      "I661.6" { ExternalVisible := 'False'} : Bool := FALSE;   // I661.6
      "I661.7" { ExternalVisible := 'False'} : Bool := FALSE;   // I661.7
      "I662.0" { ExternalVisible := 'False'} : Bool := FALSE;   // I662.0
      "I662.1" { ExternalVisible := 'False'} : Bool := FALSE;   // I662.1
      "I662.2" { ExternalVisible := 'False'} : Bool := FALSE;   // I662.2
      "I662.3" { ExternalVisible := 'False'} : Bool := FALSE;   // I662.3
      "I662.4" { ExternalVisible := 'False'} : Bool := FALSE;   // I662.4
      "I662.5" { ExternalVisible := 'False'} : Bool := FALSE;   // I662.5
      "I662.6" { ExternalVisible := 'False'} : Bool := FALSE;   // I662.6
      "I662.7" { ExternalVisible := 'False'} : Bool := FALSE;   // I662.7
      "I663.0" { ExternalVisible := 'False'} : Bool := FALSE;   // I663.0
      "I663.1" { ExternalVisible := 'False'} : Bool := FALSE;   // I663.1
      "I663.2" { ExternalVisible := 'False'} : Bool := FALSE;   // I663.2
      "I663.3" { ExternalVisible := 'False'} : Bool := FALSE;   // I663.3
      "I663.4" { ExternalVisible := 'False'} : Bool := FALSE;   // I663.4
      "I663.5" { ExternalVisible := 'False'} : Bool := FALSE;   // I663.5
      "I663.6" { ExternalVisible := 'False'} : Bool := FALSE;   // I663.6
      "I663.7" { ExternalVisible := 'False'} : Bool := FALSE;   // I663.7
      "I664.0" { ExternalVisible := 'False'} : Bool := FALSE;   // I664.0
      "I664.1" { ExternalVisible := 'False'} : Bool := FALSE;   // I664.1
      "I664.2" { ExternalVisible := 'False'} : Bool := FALSE;   // I664.2
      "I664.3" { ExternalVisible := 'False'} : Bool := FALSE;   // I664.3
      "I664.4" { ExternalVisible := 'False'} : Bool := FALSE;   // I664.4
      "I664.5" { ExternalVisible := 'False'} : Bool := FALSE;   // I664.5
      "I664.6" { ExternalVisible := 'False'} : Bool := FALSE;   // I664.6
      "I664.7" { ExternalVisible := 'False'} : Bool := FALSE;   // I664.7
      "I665.0" { ExternalVisible := 'False'} : Bool := FALSE;   // I665.0
      "I665.1" { ExternalVisible := 'False'} : Bool := FALSE;   // I665.1
      "I665.2" { ExternalVisible := 'False'} : Bool := FALSE;   // I665.2
      "I665.3" { ExternalVisible := 'False'} : Bool := FALSE;   // I665.3
      "I665.4" { ExternalVisible := 'False'} : Bool := FALSE;   // I665.4
      "I665.5" { ExternalVisible := 'False'} : Bool := FALSE;   // I665.5
      "I665.6" { ExternalVisible := 'False'} : Bool := FALSE;   // I665.6
      "I665.7" { ExternalVisible := 'False'} : Bool := FALSE;   // I665.7
      "I666.0" { ExternalVisible := 'False'} : Bool := FALSE;   // I666.0
      "I666.1" { ExternalVisible := 'False'} : Bool := FALSE;   // I666.1
      "I666.2" { ExternalVisible := 'False'} : Bool := FALSE;   // I666.2
      "I666.3" { ExternalVisible := 'False'} : Bool := FALSE;   // I666.3
      "I666.4" { ExternalVisible := 'False'} : Bool := FALSE;   // I666.4
      "I666.5" { ExternalVisible := 'False'} : Bool := FALSE;   // I666.5
      "I666.6" { ExternalVisible := 'False'} : Bool := FALSE;   // I666.6
      "I666.7" { ExternalVisible := 'False'} : Bool := FALSE;   // I666.7
      "I667.0" { ExternalVisible := 'False'} : Bool := FALSE;   // I667.0
      "I667.1" { ExternalVisible := 'False'} : Bool := FALSE;   // I667.1
      "I667.2" { ExternalVisible := 'False'} : Bool := FALSE;   // I667.2
      "I667.3" { ExternalVisible := 'False'} : Bool := FALSE;   // I667.3
      "I667.4" { ExternalVisible := 'False'} : Bool := FALSE;   // I667.4
      "I667.5" { ExternalVisible := 'False'} : Bool := FALSE;   // I667.5
      "I667.6" { ExternalVisible := 'False'} : Bool := FALSE;   // I667.6
      "I667.7" { ExternalVisible := 'False'} : Bool := FALSE;   // I667.7
      "I668.0" { ExternalVisible := 'False'} : Bool := FALSE;   // I668.0
      "I668.1" { ExternalVisible := 'False'} : Bool := FALSE;   // I668.1
      "I668.2" { ExternalVisible := 'False'} : Bool := FALSE;   // I668.2
      "I668.3" { ExternalVisible := 'False'} : Bool := FALSE;   // I668.3
      "I668.4" { ExternalVisible := 'False'} : Bool := FALSE;   // I668.4
      "I668.5" { ExternalVisible := 'False'} : Bool := FALSE;   // I668.5
      "I668.6" { ExternalVisible := 'False'} : Bool := FALSE;   // I668.6
      "I668.7" { ExternalVisible := 'False'} : Bool := FALSE;   // I668.7
      "I669.0" { ExternalVisible := 'False'} : Bool := FALSE;   // I669.0
      "I669.1" { ExternalVisible := 'False'} : Bool := FALSE;   // I669.1
      "I669.2" { ExternalVisible := 'False'} : Bool := FALSE;   // I669.2
      "I669.3" { ExternalVisible := 'False'} : Bool := FALSE;   // I669.3
      "I669.4" { ExternalVisible := 'False'} : Bool := FALSE;   // I669.4
      "I669.5" { ExternalVisible := 'False'} : Bool := FALSE;   // I669.5
      "I669.6" { ExternalVisible := 'False'} : Bool := FALSE;   // I669.6
      "I669.7" { ExternalVisible := 'False'} : Bool := FALSE;   // I669.7
      "I670.0" { ExternalVisible := 'False'} : Bool := FALSE;   // I670.0
      "I670.1" { ExternalVisible := 'False'} : Bool := FALSE;   // I670.1
      "I670.2" { ExternalVisible := 'False'} : Bool := FALSE;   // I670.2
      "I670.3" { ExternalVisible := 'False'} : Bool := FALSE;   // I670.3
      "I670.4" { ExternalVisible := 'False'} : Bool := FALSE;   // I670.4
      "I670.5" { ExternalVisible := 'False'} : Bool := FALSE;   // I670.5
      "I670.6" { ExternalVisible := 'False'} : Bool := FALSE;   // I670.6
      "I670.7" { ExternalVisible := 'False'} : Bool := FALSE;   // I670.7
      "I671.0" { ExternalVisible := 'False'} : Bool := FALSE;   // I671.0
      "I671.1" { ExternalVisible := 'False'} : Bool := FALSE;   // I671.1
      "I671.2" { ExternalVisible := 'False'} : Bool := FALSE;   // I671.2
      "I671.3" { ExternalVisible := 'False'} : Bool := FALSE;   // I671.3
      "I671.4" { ExternalVisible := 'False'} : Bool := FALSE;   // I671.4
      "I671.5" { ExternalVisible := 'False'} : Bool := FALSE;   // I671.5
      "I671.6" { ExternalVisible := 'False'} : Bool := FALSE;   // I671.6
      "I671.7" { ExternalVisible := 'False'} : Bool := FALSE;   // I671.7
      "I672.0" { ExternalVisible := 'False'} : Bool := FALSE;   // I672.0
      "I672.1" { ExternalVisible := 'False'} : Bool := FALSE;   // I672.1
      "I672.2" { ExternalVisible := 'False'} : Bool := FALSE;   // I672.2
      "I672.3" { ExternalVisible := 'False'} : Bool := FALSE;   // I672.3
      "I672.4" { ExternalVisible := 'False'} : Bool := FALSE;   // I672.4
      "I672.5" { ExternalVisible := 'False'} : Bool := FALSE;   // I672.5
      "I672.6" { ExternalVisible := 'False'} : Bool := FALSE;   // I672.6
      "I672.7" { ExternalVisible := 'False'} : Bool := FALSE;   // I672.7
      "I673.0" { ExternalVisible := 'False'} : Bool := FALSE;   // I673.0
      "I673.1" { ExternalVisible := 'False'} : Bool := FALSE;   // I673.1
      "I673.2" { ExternalVisible := 'False'} : Bool := FALSE;   // I673.2
      "I673.3" { ExternalVisible := 'False'} : Bool := FALSE;   // I673.3
      "I673.4" { ExternalVisible := 'False'} : Bool := FALSE;   // I673.4
      "I673.5" { ExternalVisible := 'False'} : Bool := FALSE;   // I673.5
      "I673.6" { ExternalVisible := 'False'} : Bool := FALSE;   // I673.6
      "I673.7" { ExternalVisible := 'False'} : Bool := FALSE;   // I673.7
      "I674.0" { ExternalVisible := 'False'} : Bool := FALSE;   // I674.0
      "I674.1" { ExternalVisible := 'False'} : Bool := FALSE;   // I674.1
      "I674.2" { ExternalVisible := 'False'} : Bool := FALSE;   // I674.2
      "I674.3" { ExternalVisible := 'False'} : Bool := FALSE;   // I674.3
      "I674.4" { ExternalVisible := 'False'} : Bool := FALSE;   // I674.4
      "I674.5" { ExternalVisible := 'False'} : Bool := FALSE;   // I674.5
      "I674.6" { ExternalVisible := 'False'} : Bool := FALSE;   // I674.6
      "I674.7" { ExternalVisible := 'False'} : Bool := FALSE;   // I674.7
      "I675.0" { ExternalVisible := 'False'} : Bool := FALSE;   // I675.0
      "I675.1" { ExternalVisible := 'False'} : Bool := FALSE;   // I675.1
      "I675.2" { ExternalVisible := 'False'} : Bool := FALSE;   // I675.2
      "I675.3" { ExternalVisible := 'False'} : Bool := FALSE;   // I675.3
      "I675.4" { ExternalVisible := 'False'} : Bool := FALSE;   // I675.4
      "I675.5" { ExternalVisible := 'False'} : Bool := FALSE;   // I675.5
      "I675.6" { ExternalVisible := 'False'} : Bool := FALSE;   // I675.6
      "I675.7" { ExternalVisible := 'False'} : Bool := FALSE;   // I675.7
      "I676.0" { ExternalVisible := 'False'} : Bool := FALSE;   // I676.0
      "I676.1" { ExternalVisible := 'False'} : Bool := FALSE;   // I676.1
      "I676.2" { ExternalVisible := 'False'} : Bool := FALSE;   // I676.2
      "I676.3" { ExternalVisible := 'False'} : Bool := FALSE;   // I676.3
      "I676.4" { ExternalVisible := 'False'} : Bool := FALSE;   // I676.4
      "I676.5" { ExternalVisible := 'False'} : Bool := FALSE;   // I676.5
      "I676.6" { ExternalVisible := 'False'} : Bool := FALSE;   // I676.6
      "I676.7" { ExternalVisible := 'False'} : Bool := FALSE;   // I676.7
      "I677.0" { ExternalVisible := 'False'} : Bool := FALSE;   // I677.0
      "I677.1" { ExternalVisible := 'False'} : Bool := FALSE;   // I677.1
      "I677.2" { ExternalVisible := 'False'} : Bool := FALSE;   // I677.2
      "I677.3" { ExternalVisible := 'False'} : Bool := FALSE;   // I677.3
      "I677.4" { ExternalVisible := 'False'} : Bool := FALSE;   // I677.4
      "I677.5" { ExternalVisible := 'False'} : Bool := FALSE;   // I677.5
      "I677.6" { ExternalVisible := 'False'} : Bool := FALSE;   // I677.6
      "I677.7" { ExternalVisible := 'False'} : Bool := FALSE;   // I677.7
      "I678.0" { ExternalVisible := 'False'} : Bool := FALSE;   // I678.0
      "I678.1" { ExternalVisible := 'False'} : Bool := FALSE;   // I678.1
      "I678.2" { ExternalVisible := 'False'} : Bool := FALSE;   // I678.2
      "I678.3" { ExternalVisible := 'False'} : Bool := FALSE;   // I678.3
      "I678.4" { ExternalVisible := 'False'} : Bool := FALSE;   // I678.4
      "I678.5" { ExternalVisible := 'False'} : Bool := FALSE;   // I678.5
      "I678.6" { ExternalVisible := 'False'} : Bool := FALSE;   // I678.6
      "I678.7" { ExternalVisible := 'False'} : Bool := FALSE;   // I678.7
      "I679.0" { ExternalVisible := 'False'} : Bool := FALSE;   // I679.0
      "I679.1" { ExternalVisible := 'False'} : Bool := FALSE;   // I679.1
      "I679.2" { ExternalVisible := 'False'} : Bool := FALSE;   // I679.2
      "I679.3" { ExternalVisible := 'False'} : Bool := FALSE;   // I679.3
      "I679.4" { ExternalVisible := 'False'} : Bool := FALSE;   // I679.4
      "I679.5" { ExternalVisible := 'False'} : Bool := FALSE;   // I679.5
      "I679.6" { ExternalVisible := 'False'} : Bool := FALSE;   // I679.6
      "I679.7" { ExternalVisible := 'False'} : Bool := FALSE;   // I679.7
      "I680.0" { ExternalVisible := 'False'} : Bool := FALSE;   // I680.0
      "I680.1" { ExternalVisible := 'False'} : Bool := FALSE;   // I680.1
      "I680.2" { ExternalVisible := 'False'} : Bool := FALSE;   // I680.2
      "I680.3" { ExternalVisible := 'False'} : Bool := FALSE;   // I680.3
      "I680.4" { ExternalVisible := 'False'} : Bool := FALSE;   // I680.4
      "I680.5" { ExternalVisible := 'False'} : Bool := FALSE;   // I680.5
      "I680.6" { ExternalVisible := 'False'} : Bool := FALSE;   // I680.6
      "I680.7" { ExternalVisible := 'False'} : Bool := FALSE;   // I680.7
      "I681.0" { ExternalVisible := 'False'} : Bool := FALSE;   // I681.0
      "I681.1" { ExternalVisible := 'False'} : Bool := FALSE;   // I681.1
      "I681.2" { ExternalVisible := 'False'} : Bool := FALSE;   // I681.2
      "I681.3" { ExternalVisible := 'False'} : Bool := FALSE;   // I681.3
      "I681.4" { ExternalVisible := 'False'} : Bool := FALSE;   // I681.4
      "I681.5" { ExternalVisible := 'False'} : Bool := FALSE;   // I681.5
      "I681.6" { ExternalVisible := 'False'} : Bool := FALSE;   // I681.6
      "I681.7" { ExternalVisible := 'False'} : Bool := FALSE;   // I681.7
      "I682.0" { ExternalVisible := 'False'} : Bool := FALSE;   // I682.0
      "I682.1" { ExternalVisible := 'False'} : Bool := FALSE;   // I682.1
      "I682.2" { ExternalVisible := 'False'} : Bool := FALSE;   // I682.2
      "I682.3" { ExternalVisible := 'False'} : Bool := FALSE;   // I682.3
      "I682.4" { ExternalVisible := 'False'} : Bool := FALSE;   // I682.4
      "I682.5" { ExternalVisible := 'False'} : Bool := FALSE;   // I682.5
      "I682.6" { ExternalVisible := 'False'} : Bool := FALSE;   // I682.6
      "I682.7" { ExternalVisible := 'False'} : Bool := FALSE;   // I682.7
      "I683.0" { ExternalVisible := 'False'} : Bool := FALSE;   // I683.0
      "I683.1" { ExternalVisible := 'False'} : Bool := FALSE;   // I683.1
      "I683.2" { ExternalVisible := 'False'} : Bool := FALSE;   // I683.2
      "I683.3" { ExternalVisible := 'False'} : Bool := FALSE;   // I683.3
      "I683.4" { ExternalVisible := 'False'} : Bool := FALSE;   // I683.4
      "I683.5" { ExternalVisible := 'False'} : Bool := FALSE;   // I683.5
      "I683.6" { ExternalVisible := 'False'} : Bool := FALSE;   // I683.6
      "I683.7" { ExternalVisible := 'False'} : Bool := FALSE;   // I683.7
      "I684.0" { ExternalVisible := 'False'} : Bool := FALSE;   // I684.0
      "I684.1" { ExternalVisible := 'False'} : Bool := FALSE;   // I684.1
      "I684.2" { ExternalVisible := 'False'} : Bool := FALSE;   // I684.2
      "I684.3" { ExternalVisible := 'False'} : Bool := FALSE;   // I684.3
      "I684.4" { ExternalVisible := 'False'} : Bool := FALSE;   // I684.4
      "I684.5" { ExternalVisible := 'False'} : Bool := FALSE;   // I684.5
      "I684.6" { ExternalVisible := 'False'} : Bool := FALSE;   // I684.6
      "I684.7" { ExternalVisible := 'False'} : Bool := FALSE;   // I684.7
      "I685.0" { ExternalVisible := 'False'} : Bool := FALSE;   // I685.0
      "I685.1" { ExternalVisible := 'False'} : Bool := FALSE;   // I685.1
      "I685.2" { ExternalVisible := 'False'} : Bool := FALSE;   // I685.2
      "I685.3" { ExternalVisible := 'False'} : Bool := FALSE;   // I685.3
      "I685.4" { ExternalVisible := 'False'} : Bool := FALSE;   // I685.4
      "I685.5" { ExternalVisible := 'False'} : Bool := FALSE;   // I685.5
      "I685.6" { ExternalVisible := 'False'} : Bool := FALSE;   // I685.6
      "I685.7" { ExternalVisible := 'False'} : Bool := FALSE;   // I685.7
      "I686.0" { ExternalVisible := 'False'} : Bool := FALSE;   // I686.0
      "I686.1" { ExternalVisible := 'False'} : Bool := FALSE;   // I686.1
      "I686.2" { ExternalVisible := 'False'} : Bool := FALSE;   // I686.2
      "I686.3" { ExternalVisible := 'False'} : Bool := FALSE;   // I686.3
      "I686.4" { ExternalVisible := 'False'} : Bool := FALSE;   // I686.4
      "I686.5" { ExternalVisible := 'False'} : Bool := FALSE;   // I686.5
      "I686.6" { ExternalVisible := 'False'} : Bool := FALSE;   // I686.6
      "I686.7" { ExternalVisible := 'False'} : Bool := FALSE;   // I686.7
      "I687.0" { ExternalVisible := 'False'} : Bool := FALSE;   // I687.0
      "I687.1" { ExternalVisible := 'False'} : Bool := FALSE;   // I687.1
      "I687.2" { ExternalVisible := 'False'} : Bool := FALSE;   // I687.2
      "I687.3" { ExternalVisible := 'False'} : Bool := FALSE;   // I687.3
      "I687.4" { ExternalVisible := 'False'} : Bool := FALSE;   // I687.4
      "I687.5" { ExternalVisible := 'False'} : Bool := FALSE;   // I687.5
      "I687.6" { ExternalVisible := 'False'} : Bool := FALSE;   // I687.6
      "I687.7" { ExternalVisible := 'False'} : Bool := FALSE;   // I687.7
      "I688.0" { ExternalVisible := 'False'} : Bool := FALSE;   // I688.0
      "I688.1" { ExternalVisible := 'False'} : Bool := FALSE;   // I688.1
      "I688.2" { ExternalVisible := 'False'} : Bool := FALSE;   // I688.2
      "I688.3" { ExternalVisible := 'False'} : Bool := FALSE;   // I688.3
      "I688.4" { ExternalVisible := 'False'} : Bool := FALSE;   // I688.4
      "I688.5" { ExternalVisible := 'False'} : Bool := FALSE;   // I688.5
      "I688.6" { ExternalVisible := 'False'} : Bool := FALSE;   // I688.6
      "I688.7" { ExternalVisible := 'False'} : Bool := FALSE;   // I688.7
      "I689.0" { ExternalVisible := 'False'} : Bool := FALSE;   // I689.0
      "I689.1" { ExternalVisible := 'False'} : Bool := FALSE;   // I689.1
      "I689.2" { ExternalVisible := 'False'} : Bool := FALSE;   // I689.2
      "I689.3" { ExternalVisible := 'False'} : Bool := FALSE;   // I689.3
      "I689.4" { ExternalVisible := 'False'} : Bool := FALSE;   // I689.4
      "I689.5" { ExternalVisible := 'False'} : Bool := FALSE;   // I689.5
      "I689.6" { ExternalVisible := 'False'} : Bool := FALSE;   // I689.6
      "I689.7" { ExternalVisible := 'False'} : Bool := FALSE;   // I689.7
      "I690.0" { ExternalVisible := 'False'} : Bool := FALSE;   // I690.0
      "I690.1" { ExternalVisible := 'False'} : Bool := FALSE;   // I690.1
      "I690.2" { ExternalVisible := 'False'} : Bool := FALSE;   // I690.2
      "I690.3" { ExternalVisible := 'False'} : Bool := FALSE;   // I690.3
      "I690.4" { ExternalVisible := 'False'} : Bool := FALSE;   // I690.4
      "I690.5" { ExternalVisible := 'False'} : Bool := FALSE;   // I690.5
      "I690.6" { ExternalVisible := 'False'} : Bool := FALSE;   // I690.6
      "I690.7" { ExternalVisible := 'False'} : Bool := FALSE;   // I690.7
      "I691.0" { ExternalVisible := 'False'} : Bool := FALSE;   // I691.0
      "I691.1" { ExternalVisible := 'False'} : Bool := FALSE;   // I691.1
      "I691.2" { ExternalVisible := 'False'} : Bool := FALSE;   // I691.2
      "I691.3" { ExternalVisible := 'False'} : Bool := FALSE;   // I691.3
      "I691.4" { ExternalVisible := 'False'} : Bool := FALSE;   // I691.4
      "I691.5" { ExternalVisible := 'False'} : Bool := FALSE;   // I691.5
      "I691.6" { ExternalVisible := 'False'} : Bool := FALSE;   // I691.6
      "I691.7" { ExternalVisible := 'False'} : Bool := FALSE;   // I691.7
      "I692.0" { ExternalVisible := 'False'} : Bool := FALSE;   // I692.0
      "I692.1" { ExternalVisible := 'False'} : Bool := FALSE;   // I692.1
      "I692.2" { ExternalVisible := 'False'} : Bool := FALSE;   // I692.2
      "I692.3" { ExternalVisible := 'False'} : Bool := FALSE;   // I692.3
      "I692.4" { ExternalVisible := 'False'} : Bool := FALSE;   // I692.4
      "I692.5" { ExternalVisible := 'False'} : Bool := FALSE;   // I692.5
      "I692.6" { ExternalVisible := 'False'} : Bool := FALSE;   // I692.6
      "I692.7" { ExternalVisible := 'False'} : Bool := FALSE;   // I692.7
      "I693.0" { ExternalVisible := 'False'} : Bool := FALSE;   // I693.0
      "I693.1" { ExternalVisible := 'False'} : Bool := FALSE;   // I693.1
      "I693.2" { ExternalVisible := 'False'} : Bool := FALSE;   // I693.2
      "I693.3" { ExternalVisible := 'False'} : Bool := FALSE;   // I693.3
      "I693.4" { ExternalVisible := 'False'} : Bool := FALSE;   // I693.4
      "I693.5" { ExternalVisible := 'False'} : Bool := FALSE;   // I693.5
      "I693.6" { ExternalVisible := 'False'} : Bool := FALSE;   // I693.6
      "I693.7" { ExternalVisible := 'False'} : Bool := FALSE;   // I693.7
      "I694.0" { ExternalVisible := 'False'} : Bool := FALSE;   // I694.0
      "I694.1" { ExternalVisible := 'False'} : Bool := FALSE;   // I694.1
      "I694.2" { ExternalVisible := 'False'} : Bool := FALSE;   // I694.2
      "I694.3" { ExternalVisible := 'False'} : Bool := FALSE;   // I694.3
      "I694.4" { ExternalVisible := 'False'} : Bool := FALSE;   // I694.4
      "I694.5" { ExternalVisible := 'False'} : Bool := FALSE;   // I694.5
      "I694.6" { ExternalVisible := 'False'} : Bool := FALSE;   // I694.6
      "I694.7" { ExternalVisible := 'False'} : Bool := FALSE;   // I694.7
      "I695.0" { ExternalVisible := 'False'} : Bool := FALSE;   // I695.0
      "I695.1" { ExternalVisible := 'False'} : Bool := FALSE;   // I695.1
      "I695.2" { ExternalVisible := 'False'} : Bool := FALSE;   // I695.2
      "I695.3" { ExternalVisible := 'False'} : Bool := FALSE;   // I695.3
      "I695.4" { ExternalVisible := 'False'} : Bool := FALSE;   // I695.4
      "I695.5" { ExternalVisible := 'False'} : Bool := FALSE;   // I695.5
      "I695.6" { ExternalVisible := 'False'} : Bool := FALSE;   // I695.6
      "I695.7" { ExternalVisible := 'False'} : Bool := FALSE;   // I695.7
      "I696.0" { ExternalVisible := 'False'} : Bool := FALSE;   // I696.0
      "I696.1" { ExternalVisible := 'False'} : Bool := FALSE;   // I696.1
      "I696.2" { ExternalVisible := 'False'} : Bool := FALSE;   // I696.2
      "I696.3" { ExternalVisible := 'False'} : Bool := FALSE;   // I696.3
      "I696.4" { ExternalVisible := 'False'} : Bool := FALSE;   // I696.4
      "I696.5" { ExternalVisible := 'False'} : Bool := FALSE;   // I696.5
      "I696.6" { ExternalVisible := 'False'} : Bool := FALSE;   // I696.6
      "I696.7" { ExternalVisible := 'False'} : Bool := FALSE;   // I696.7
      "I697.0" { ExternalVisible := 'False'} : Bool := FALSE;   // I697.0
      "I697.1" { ExternalVisible := 'False'} : Bool := FALSE;   // I697.1
      "I697.2" { ExternalVisible := 'False'} : Bool := FALSE;   // I697.2
      "I697.3" { ExternalVisible := 'False'} : Bool := FALSE;   // I697.3
      "I697.4" { ExternalVisible := 'False'} : Bool := FALSE;   // I697.4
      "I697.5" { ExternalVisible := 'False'} : Bool := FALSE;   // I697.5
      "I697.6" { ExternalVisible := 'False'} : Bool := FALSE;   // I697.6
      "I697.7" { ExternalVisible := 'False'} : Bool := FALSE;   // I697.7
      "I698.0" { ExternalVisible := 'False'} : Bool := FALSE;   // I698.0
      "I698.1" { ExternalVisible := 'False'} : Bool := FALSE;   // I698.1
      "I698.2" { ExternalVisible := 'False'} : Bool := FALSE;   // I698.2
      "I698.3" { ExternalVisible := 'False'} : Bool := FALSE;   // I698.3
      "I698.4" { ExternalVisible := 'False'} : Bool := FALSE;   // I698.4
      "I698.5" { ExternalVisible := 'False'} : Bool := FALSE;   // I698.5
      "I698.6" { ExternalVisible := 'False'} : Bool := FALSE;   // I698.6
      "I698.7" { ExternalVisible := 'False'} : Bool := FALSE;   // I698.7
      "I699.0" { ExternalVisible := 'False'} : Bool := FALSE;   // I699.0
      "I699.1" { ExternalVisible := 'False'} : Bool := FALSE;   // I699.1
      "I699.2" { ExternalVisible := 'False'} : Bool := FALSE;   // I699.2
      "I699.3" { ExternalVisible := 'False'} : Bool := FALSE;   // I699.3
      "I699.4" { ExternalVisible := 'False'} : Bool := FALSE;   // I699.4
      "I699.5" { ExternalVisible := 'False'} : Bool := FALSE;   // I699.5
      "I699.6" { ExternalVisible := 'False'} : Bool := FALSE;   // I699.6
      "I699.7" { ExternalVisible := 'False'} : Bool := FALSE;   // I699.7
      "I700.0" { ExternalVisible := 'False'} : Bool := FALSE;   // I700.0
      "I700.1" { ExternalVisible := 'False'} : Bool := FALSE;   // I700.1
      "I700.2" { ExternalVisible := 'False'} : Bool := FALSE;   // I700.2
      "I700.3" { ExternalVisible := 'False'} : Bool := FALSE;   // I700.3
      "I700.4" { ExternalVisible := 'False'} : Bool := FALSE;   // I700.4
      "I700.5" { ExternalVisible := 'False'} : Bool := FALSE;   // I700.5
      "I700.6" { ExternalVisible := 'False'} : Bool := FALSE;   // I700.6
      "I700.7" { ExternalVisible := 'False'} : Bool := FALSE;   // I700.7
      "I701.0" { ExternalVisible := 'False'} : Bool := FALSE;   // I701.0
      "I701.1" { ExternalVisible := 'False'} : Bool := FALSE;   // I701.1
      "I701.2" { ExternalVisible := 'False'} : Bool := FALSE;   // I701.2
      "I701.3" { ExternalVisible := 'False'} : Bool := FALSE;   // I701.3
      "I701.4" { ExternalVisible := 'False'} : Bool := FALSE;   // I701.4
      "I701.5" { ExternalVisible := 'False'} : Bool := FALSE;   // I701.5
      "I701.6" { ExternalVisible := 'False'} : Bool := FALSE;   // I701.6
      "I701.7" { ExternalVisible := 'False'} : Bool := FALSE;   // I701.7
      "I702.0" { ExternalVisible := 'False'} : Bool := FALSE;   // I702.0
      "I702.1" { ExternalVisible := 'False'} : Bool := FALSE;   // I702.1
      "I702.2" { ExternalVisible := 'False'} : Bool := FALSE;   // I702.2
      "I702.3" { ExternalVisible := 'False'} : Bool := FALSE;   // I702.3
      "I702.4" { ExternalVisible := 'False'} : Bool := FALSE;   // I702.4
      "I702.5" { ExternalVisible := 'False'} : Bool := FALSE;   // I702.5
      "I702.6" { ExternalVisible := 'False'} : Bool := FALSE;   // I702.6
      "I702.7" { ExternalVisible := 'False'} : Bool := FALSE;   // I702.7
      "I703.0" { ExternalVisible := 'False'} : Bool := FALSE;   // I703.0
      "I703.1" { ExternalVisible := 'False'} : Bool := FALSE;   // I703.1
      "I703.2" { ExternalVisible := 'False'} : Bool := FALSE;   // I703.2
      "I703.3" { ExternalVisible := 'False'} : Bool := FALSE;   // I703.3
      "I703.4" { ExternalVisible := 'False'} : Bool := FALSE;   // I703.4
      "I703.5" { ExternalVisible := 'False'} : Bool := FALSE;   // I703.5
      "I703.6" { ExternalVisible := 'False'} : Bool := FALSE;   // I703.6
      "I703.7" { ExternalVisible := 'False'} : Bool := FALSE;   // I703.7
      "I704.0" { ExternalVisible := 'False'} : Bool := FALSE;   // I704.0
      "I704.1" { ExternalVisible := 'False'} : Bool := FALSE;   // I704.1
      "I704.2" { ExternalVisible := 'False'} : Bool := FALSE;   // I704.2
      "I704.3" { ExternalVisible := 'False'} : Bool := FALSE;   // I704.3
      "I704.4" { ExternalVisible := 'False'} : Bool := FALSE;   // I704.4
      "I704.5" { ExternalVisible := 'False'} : Bool := FALSE;   // I704.5
      "I704.6" { ExternalVisible := 'False'} : Bool := FALSE;   // I704.6
      "I704.7" { ExternalVisible := 'False'} : Bool := FALSE;   // I704.7
      "I705.0" { ExternalVisible := 'False'} : Bool := FALSE;   // I705.0
      "I705.1" { ExternalVisible := 'False'} : Bool := FALSE;   // I705.1
      "I705.2" { ExternalVisible := 'False'} : Bool := FALSE;   // I705.2
      "I705.3" { ExternalVisible := 'False'} : Bool := FALSE;   // I705.3
      "I705.4" { ExternalVisible := 'False'} : Bool := FALSE;   // I705.4
      "I705.5" { ExternalVisible := 'False'} : Bool := FALSE;   // I705.5
      "I705.6" { ExternalVisible := 'False'} : Bool := FALSE;   // I705.6
      "I705.7" { ExternalVisible := 'False'} : Bool := FALSE;   // I705.7
      "I706.0" { ExternalVisible := 'False'} : Bool := FALSE;   // I706.0
      "I706.1" { ExternalVisible := 'False'} : Bool := FALSE;   // I706.1
      "I706.2" { ExternalVisible := 'False'} : Bool := FALSE;   // I706.2
      "I706.3" { ExternalVisible := 'False'} : Bool := FALSE;   // I706.3
      "I706.4" { ExternalVisible := 'False'} : Bool := FALSE;   // I706.4
      "I706.5" { ExternalVisible := 'False'} : Bool := FALSE;   // I706.5
      "I706.6" { ExternalVisible := 'False'} : Bool := FALSE;   // I706.6
      "I706.7" { ExternalVisible := 'False'} : Bool := FALSE;   // I706.7
      "I707.0" { ExternalVisible := 'False'} : Bool := FALSE;   // I707.0
      "I707.1" { ExternalVisible := 'False'} : Bool := FALSE;   // I707.1
      "I707.2" { ExternalVisible := 'False'} : Bool := FALSE;   // I707.2
      "I707.3" { ExternalVisible := 'False'} : Bool := FALSE;   // I707.3
      "I707.4" { ExternalVisible := 'False'} : Bool := FALSE;   // I707.4
      "I707.5" { ExternalVisible := 'False'} : Bool := FALSE;   // I707.5
      "I707.6" { ExternalVisible := 'False'} : Bool := FALSE;   // I707.6
      "I707.7" { ExternalVisible := 'False'} : Bool := FALSE;   // I707.7
      "I708.0" { ExternalVisible := 'False'} : Bool := FALSE;   // I708.0
      "I708.1" { ExternalVisible := 'False'} : Bool := FALSE;   // I708.1
      "I708.2" { ExternalVisible := 'False'} : Bool := FALSE;   // I708.2
      "I708.3" { ExternalVisible := 'False'} : Bool := FALSE;   // I708.3
      "I708.4" { ExternalVisible := 'False'} : Bool := FALSE;   // I708.4
      "I708.5" { ExternalVisible := 'False'} : Bool := FALSE;   // I708.5
      "I708.6" { ExternalVisible := 'False'} : Bool := FALSE;   // I708.6
      "I708.7" { ExternalVisible := 'False'} : Bool := FALSE;   // I708.7
      "I709.0" { ExternalVisible := 'False'} : Bool := FALSE;   // I709.0
      "I709.1" { ExternalVisible := 'False'} : Bool := FALSE;   // I709.1
      "I709.2" { ExternalVisible := 'False'} : Bool := FALSE;   // I709.2
      "I709.3" { ExternalVisible := 'False'} : Bool := FALSE;   // I709.3
      "I709.4" { ExternalVisible := 'False'} : Bool := FALSE;   // I709.4
      "I709.5" { ExternalVisible := 'False'} : Bool := FALSE;   // I709.5
      "I709.6" { ExternalVisible := 'False'} : Bool := FALSE;   // I709.6
      "I709.7" { ExternalVisible := 'False'} : Bool := FALSE;   // I709.7
      "I710.0" { ExternalVisible := 'False'} : Bool := FALSE;   // I710.0
      "I710.1" { ExternalVisible := 'False'} : Bool := FALSE;   // I710.1
      "I710.2" { ExternalVisible := 'False'} : Bool := FALSE;   // I710.2
      "I710.3" { ExternalVisible := 'False'} : Bool := FALSE;   // I710.3
      "I710.4" { ExternalVisible := 'False'} : Bool := FALSE;   // I710.4
      "I710.5" { ExternalVisible := 'False'} : Bool := FALSE;   // I710.5
      "I710.6" { ExternalVisible := 'False'} : Bool := FALSE;   // I710.6
      "I710.7" { ExternalVisible := 'False'} : Bool := FALSE;   // I710.7
      "I711.0" { ExternalVisible := 'False'} : Bool := FALSE;   // I711.0
      "I711.1" { ExternalVisible := 'False'} : Bool := FALSE;   // I711.1
      "I711.2" { ExternalVisible := 'False'} : Bool := FALSE;   // I711.2
      "I711.3" { ExternalVisible := 'False'} : Bool := FALSE;   // I711.3
      "I711.4" { ExternalVisible := 'False'} : Bool := FALSE;   // I711.4
      "I711.5" { ExternalVisible := 'False'} : Bool := FALSE;   // I711.5
      "I711.6" { ExternalVisible := 'False'} : Bool := FALSE;   // I711.6
      "I711.7" { ExternalVisible := 'False'} : Bool := FALSE;   // I711.7
      "I712.0" { ExternalVisible := 'False'} : Bool := FALSE;   // I712.0
      "I712.1" { ExternalVisible := 'False'} : Bool := FALSE;   // I712.1
      "I712.2" { ExternalVisible := 'False'} : Bool := FALSE;   // I712.2
      "I712.3" { ExternalVisible := 'False'} : Bool := FALSE;   // I712.3
      "I712.4" { ExternalVisible := 'False'} : Bool := FALSE;   // I712.4
      "I712.5" { ExternalVisible := 'False'} : Bool := FALSE;   // I712.5
      "I712.6" { ExternalVisible := 'False'} : Bool := FALSE;   // I712.6
      "I712.7" { ExternalVisible := 'False'} : Bool := FALSE;   // I712.7
      "I713.0" { ExternalVisible := 'False'} : Bool := FALSE;   // I713.0
      "I713.1" { ExternalVisible := 'False'} : Bool := FALSE;   // I713.1
      "I713.2" { ExternalVisible := 'False'} : Bool := FALSE;   // I713.2
      "I713.3" { ExternalVisible := 'False'} : Bool := FALSE;   // I713.3
      "I713.4" { ExternalVisible := 'False'} : Bool := FALSE;   // I713.4
      "I713.5" { ExternalVisible := 'False'} : Bool := FALSE;   // I713.5
      "I713.6" { ExternalVisible := 'False'} : Bool := FALSE;   // I713.6
      "I713.7" { ExternalVisible := 'False'} : Bool := FALSE;   // I713.7
      "I714.0" { ExternalVisible := 'False'} : Bool := FALSE;   // I714.0
      "I714.1" { ExternalVisible := 'False'} : Bool := FALSE;   // I714.1
      "I714.2" { ExternalVisible := 'False'} : Bool := FALSE;   // I714.2
      "I714.3" { ExternalVisible := 'False'} : Bool := FALSE;   // I714.3
      "I714.4" { ExternalVisible := 'False'} : Bool := FALSE;   // I714.4
      "I714.5" { ExternalVisible := 'False'} : Bool := FALSE;   // I714.5
      "I714.6" { ExternalVisible := 'False'} : Bool := FALSE;   // I714.6
      "I714.7" { ExternalVisible := 'False'} : Bool := FALSE;   // I714.7
      "I715.0" { ExternalVisible := 'False'} : Bool := FALSE;   // I715.0
      "I715.1" { ExternalVisible := 'False'} : Bool := FALSE;   // I715.1
      "I715.2" { ExternalVisible := 'False'} : Bool := FALSE;   // I715.2
      "I715.3" { ExternalVisible := 'False'} : Bool := FALSE;   // I715.3
      "I715.4" { ExternalVisible := 'False'} : Bool := FALSE;   // I715.4
      "I715.5" { ExternalVisible := 'False'} : Bool := FALSE;   // I715.5
      "I715.6" { ExternalVisible := 'False'} : Bool := FALSE;   // I715.6
      "I715.7" { ExternalVisible := 'False'} : Bool := FALSE;   // I715.7
      "I716.0" { ExternalVisible := 'False'} : Bool := FALSE;   // I716.0
      "I716.1" { ExternalVisible := 'False'} : Bool := FALSE;   // I716.1
      "I716.2" { ExternalVisible := 'False'} : Bool := FALSE;   // I716.2
      "I716.3" { ExternalVisible := 'False'} : Bool := FALSE;   // I716.3
      "I716.4" { ExternalVisible := 'False'} : Bool := FALSE;   // I716.4
      "I716.5" { ExternalVisible := 'False'} : Bool := FALSE;   // I716.5
      "I716.6" { ExternalVisible := 'False'} : Bool := FALSE;   // I716.6
      "I716.7" { ExternalVisible := 'False'} : Bool := FALSE;   // I716.7
      "I717.0" { ExternalVisible := 'False'} : Bool := FALSE;   // I717.0
      "I717.1" { ExternalVisible := 'False'} : Bool := FALSE;   // I717.1
      "I717.2" { ExternalVisible := 'False'} : Bool := FALSE;   // I717.2
      "I717.3" { ExternalVisible := 'False'} : Bool := FALSE;   // I717.3
      "I717.4" { ExternalVisible := 'False'} : Bool := FALSE;   // I717.4
      "I717.5" { ExternalVisible := 'False'} : Bool := FALSE;   // I717.5
      "I717.6" { ExternalVisible := 'False'} : Bool := FALSE;   // I717.6
      "I717.7" { ExternalVisible := 'False'} : Bool := FALSE;   // I717.7
      "I718.0" { ExternalVisible := 'False'} : Bool := FALSE;   // I718.0
      "I718.1" { ExternalVisible := 'False'} : Bool := FALSE;   // I718.1
      "I718.2" { ExternalVisible := 'False'} : Bool := FALSE;   // I718.2
      "I718.3" { ExternalVisible := 'False'} : Bool := FALSE;   // I718.3
      "I718.4" { ExternalVisible := 'False'} : Bool := FALSE;   // I718.4
      "I718.5" { ExternalVisible := 'False'} : Bool := FALSE;   // I718.5
      "I718.6" { ExternalVisible := 'False'} : Bool := FALSE;   // I718.6
      "I718.7" { ExternalVisible := 'False'} : Bool := FALSE;   // I718.7
      "I719.0" { ExternalVisible := 'False'} : Bool := FALSE;   // I719.0
      "I719.1" { ExternalVisible := 'False'} : Bool := FALSE;   // I719.1
      "I719.2" { ExternalVisible := 'False'} : Bool := FALSE;   // I719.2
      "I719.3" { ExternalVisible := 'False'} : Bool := FALSE;   // I719.3
      "I719.4" { ExternalVisible := 'False'} : Bool := FALSE;   // I719.4
      "I719.5" { ExternalVisible := 'False'} : Bool := FALSE;   // I719.5
      "I719.6" { ExternalVisible := 'False'} : Bool := FALSE;   // I719.6
      "I719.7" { ExternalVisible := 'False'} : Bool := FALSE;   // I719.7
      "I720.0" { ExternalVisible := 'False'} : Bool := FALSE;   // I720.0
      "I720.1" { ExternalVisible := 'False'} : Bool := FALSE;   // I720.1
      "I720.2" { ExternalVisible := 'False'} : Bool := FALSE;   // I720.2
      "I720.3" { ExternalVisible := 'False'} : Bool := FALSE;   // I720.3
      "I720.4" { ExternalVisible := 'False'} : Bool := FALSE;   // I720.4
      "I720.5" { ExternalVisible := 'False'} : Bool := FALSE;   // I720.5
      "I720.6" { ExternalVisible := 'False'} : Bool := FALSE;   // I720.6
      "I720.7" { ExternalVisible := 'False'} : Bool := FALSE;   // I720.7
      "I721.0" { ExternalVisible := 'False'} : Bool := FALSE;   // I721.0
      "I721.1" { ExternalVisible := 'False'} : Bool := FALSE;   // I721.1
      "I721.2" { ExternalVisible := 'False'} : Bool := FALSE;   // I721.2
      "I721.3" { ExternalVisible := 'False'} : Bool := FALSE;   // I721.3
      "I721.4" { ExternalVisible := 'False'} : Bool := FALSE;   // I721.4
      "I721.5" { ExternalVisible := 'False'} : Bool := FALSE;   // I721.5
      "I721.6" { ExternalVisible := 'False'} : Bool := FALSE;   // I721.6
      "I721.7" { ExternalVisible := 'False'} : Bool := FALSE;   // I721.7
      "I722.0" { ExternalVisible := 'False'} : Bool := FALSE;   // I722.0
      "I722.1" { ExternalVisible := 'False'} : Bool := FALSE;   // I722.1
      "I722.2" { ExternalVisible := 'False'} : Bool := FALSE;   // I722.2
      "I722.3" { ExternalVisible := 'False'} : Bool := FALSE;   // I722.3
      "I722.4" { ExternalVisible := 'False'} : Bool := FALSE;   // I722.4
      "I722.5" { ExternalVisible := 'False'} : Bool := FALSE;   // I722.5
      "I722.6" { ExternalVisible := 'False'} : Bool := FALSE;   // I722.6
      "I722.7" { ExternalVisible := 'False'} : Bool := FALSE;   // I722.7
      "I723.0" { ExternalVisible := 'False'} : Bool := FALSE;   // I723.0
      "I723.1" { ExternalVisible := 'False'} : Bool := FALSE;   // I723.1
      "I723.2" { ExternalVisible := 'False'} : Bool := FALSE;   // I723.2
      "I723.3" { ExternalVisible := 'False'} : Bool := FALSE;   // I723.3
      "I723.4" { ExternalVisible := 'False'} : Bool := FALSE;   // I723.4
      "I723.5" { ExternalVisible := 'False'} : Bool := FALSE;   // I723.5
      "I723.6" { ExternalVisible := 'False'} : Bool := FALSE;   // I723.6
      "I723.7" { ExternalVisible := 'False'} : Bool := FALSE;   // I723.7
      "I724.0" { ExternalVisible := 'False'} : Bool := FALSE;   // I724.0
      "I724.1" { ExternalVisible := 'False'} : Bool := FALSE;   // I724.1
      "I724.2" { ExternalVisible := 'False'} : Bool := FALSE;   // I724.2
      "I724.3" { ExternalVisible := 'False'} : Bool := FALSE;   // I724.3
      "I724.4" { ExternalVisible := 'False'} : Bool := FALSE;   // I724.4
      "I724.5" { ExternalVisible := 'False'} : Bool := FALSE;   // I724.5
      "I724.6" { ExternalVisible := 'False'} : Bool := FALSE;   // I724.6
      "I724.7" { ExternalVisible := 'False'} : Bool := FALSE;   // I724.7
      "I725.0" { ExternalVisible := 'False'} : Bool := FALSE;   // I725.0
      "I725.1" { ExternalVisible := 'False'} : Bool := FALSE;   // I725.1
      "I725.2" { ExternalVisible := 'False'} : Bool := FALSE;   // I725.2
      "I725.3" { ExternalVisible := 'False'} : Bool := FALSE;   // I725.3
      "I725.4" { ExternalVisible := 'False'} : Bool := FALSE;   // I725.4
      "I725.5" { ExternalVisible := 'False'} : Bool := FALSE;   // I725.5
      "I725.6" { ExternalVisible := 'False'} : Bool := FALSE;   // I725.6
      "I725.7" { ExternalVisible := 'False'} : Bool := FALSE;   // I725.7
      "I726.0" { ExternalVisible := 'False'} : Bool := FALSE;   // I726.0
      "I726.1" { ExternalVisible := 'False'} : Bool := FALSE;   // I726.1
      "I726.2" { ExternalVisible := 'False'} : Bool := FALSE;   // I726.2
      "I726.3" { ExternalVisible := 'False'} : Bool := FALSE;   // I726.3
      "I726.4" { ExternalVisible := 'False'} : Bool := FALSE;   // I726.4
      "I726.5" { ExternalVisible := 'False'} : Bool := FALSE;   // I726.5
      "I726.6" { ExternalVisible := 'False'} : Bool := FALSE;   // I726.6
      "I726.7" { ExternalVisible := 'False'} : Bool := FALSE;   // I726.7
      "I727.0" { ExternalVisible := 'False'} : Bool := FALSE;   // I727.0
      "I727.1" { ExternalVisible := 'False'} : Bool := FALSE;   // I727.1
      "I727.2" { ExternalVisible := 'False'} : Bool := FALSE;   // I727.2
      "I727.3" { ExternalVisible := 'False'} : Bool := FALSE;   // I727.3
      "I727.4" { ExternalVisible := 'False'} : Bool := FALSE;   // I727.4
      "I727.5" { ExternalVisible := 'False'} : Bool := FALSE;   // I727.5
      "I727.6" { ExternalVisible := 'False'} : Bool := FALSE;   // I727.6
      "I727.7" { ExternalVisible := 'False'} : Bool := FALSE;   // I727.7
      "I728.0" { ExternalVisible := 'False'} : Bool := FALSE;   // I728.0
      "I728.1" { ExternalVisible := 'False'} : Bool := FALSE;   // I728.1
      "I728.2" { ExternalVisible := 'False'} : Bool := FALSE;   // I728.2
      "I728.3" { ExternalVisible := 'False'} : Bool := FALSE;   // I728.3
      "I728.4" { ExternalVisible := 'False'} : Bool := FALSE;   // I728.4
      "I728.5" { ExternalVisible := 'False'} : Bool := FALSE;   // I728.5
      "I728.6" { ExternalVisible := 'False'} : Bool := FALSE;   // I728.6
      "I728.7" { ExternalVisible := 'False'} : Bool := FALSE;   // I728.7
      "I729.0" { ExternalVisible := 'False'} : Bool := FALSE;   // I729.0
      "I729.1" { ExternalVisible := 'False'} : Bool := FALSE;   // I729.1
      "I729.2" { ExternalVisible := 'False'} : Bool := FALSE;   // I729.2
      "I729.3" { ExternalVisible := 'False'} : Bool := FALSE;   // I729.3
      "I729.4" { ExternalVisible := 'False'} : Bool := FALSE;   // I729.4
      "I729.5" { ExternalVisible := 'False'} : Bool := FALSE;   // I729.5
      "I729.6" { ExternalVisible := 'False'} : Bool := FALSE;   // I729.6
      "I729.7" { ExternalVisible := 'False'} : Bool := FALSE;   // I729.7
      "I730.0" { ExternalVisible := 'False'} : Bool := FALSE;   // I730.0
      "I730.1" { ExternalVisible := 'False'} : Bool := FALSE;   // I730.1
      "I730.2" { ExternalVisible := 'False'} : Bool := FALSE;   // I730.2
      "I730.3" { ExternalVisible := 'False'} : Bool := FALSE;   // I730.3
      "I730.4" { ExternalVisible := 'False'} : Bool := FALSE;   // I730.4
      "I730.5" { ExternalVisible := 'False'} : Bool := FALSE;   // I730.5
      "I730.6" { ExternalVisible := 'False'} : Bool := FALSE;   // I730.6
      "I730.7" { ExternalVisible := 'False'} : Bool := FALSE;   // I730.7
      "I731.0" { ExternalVisible := 'False'} : Bool := FALSE;   // I731.0
      "I731.1" { ExternalVisible := 'False'} : Bool := FALSE;   // I731.1
      "I731.2" { ExternalVisible := 'False'} : Bool := FALSE;   // I731.2
      "I731.3" { ExternalVisible := 'False'} : Bool := FALSE;   // I731.3
      "I731.4" { ExternalVisible := 'False'} : Bool := FALSE;   // I731.4
      "I731.5" { ExternalVisible := 'False'} : Bool := FALSE;   // I731.5
      "I731.6" { ExternalVisible := 'False'} : Bool := FALSE;   // I731.6
      "I731.7" { ExternalVisible := 'False'} : Bool := FALSE;   // I731.7
      "I732.0" { ExternalVisible := 'False'} : Bool := FALSE;   // I732.0
      "I732.1" { ExternalVisible := 'False'} : Bool := FALSE;   // I732.1
      "I732.2" { ExternalVisible := 'False'} : Bool := FALSE;   // I732.2
      "I732.3" { ExternalVisible := 'False'} : Bool := FALSE;   // I732.3
      "I732.4" { ExternalVisible := 'False'} : Bool := FALSE;   // I732.4
      "I732.5" { ExternalVisible := 'False'} : Bool := FALSE;   // I732.5
      "I732.6" { ExternalVisible := 'False'} : Bool := FALSE;   // I732.6
      "I732.7" { ExternalVisible := 'False'} : Bool := FALSE;   // I732.7
      "I733.0" { ExternalVisible := 'False'} : Bool := FALSE;   // I733.0
      "I733.1" { ExternalVisible := 'False'} : Bool := FALSE;   // I733.1
      "I733.2" { ExternalVisible := 'False'} : Bool := FALSE;   // I733.2
      "I733.3" { ExternalVisible := 'False'} : Bool := FALSE;   // I733.3
      "I733.4" { ExternalVisible := 'False'} : Bool := FALSE;   // I733.4
      "I733.5" { ExternalVisible := 'False'} : Bool := FALSE;   // I733.5
      "I733.6" { ExternalVisible := 'False'} : Bool := FALSE;   // I733.6
      "I733.7" { ExternalVisible := 'False'} : Bool := FALSE;   // I733.7
      "I734.0" { ExternalVisible := 'False'} : Bool := FALSE;   // I734.0
      "I734.1" { ExternalVisible := 'False'} : Bool := FALSE;   // I734.1
      "I734.2" { ExternalVisible := 'False'} : Bool := FALSE;   // I734.2
      "I734.3" { ExternalVisible := 'False'} : Bool := FALSE;   // I734.3
      "I734.4" { ExternalVisible := 'False'} : Bool := FALSE;   // I734.4
      "I734.5" { ExternalVisible := 'False'} : Bool := FALSE;   // I734.5
      "I734.6" { ExternalVisible := 'False'} : Bool := FALSE;   // I734.6
      "I734.7" { ExternalVisible := 'False'} : Bool := FALSE;   // I734.7
      "I735.0" { ExternalVisible := 'False'} : Bool := FALSE;   // I735.0
      "I735.1" { ExternalVisible := 'False'} : Bool := FALSE;   // I735.1
      "I735.2" { ExternalVisible := 'False'} : Bool := FALSE;   // I735.2
      "I735.3" { ExternalVisible := 'False'} : Bool := FALSE;   // I735.3
      "I735.4" { ExternalVisible := 'False'} : Bool := FALSE;   // I735.4
      "I735.5" { ExternalVisible := 'False'} : Bool := FALSE;   // I735.5
      "I735.6" { ExternalVisible := 'False'} : Bool := FALSE;   // I735.6
      "I735.7" { ExternalVisible := 'False'} : Bool := FALSE;   // I735.7
      "I736.0" { ExternalVisible := 'False'} : Bool := FALSE;   // I736.0
      "I736.1" { ExternalVisible := 'False'} : Bool := FALSE;   // I736.1
      "I736.2" { ExternalVisible := 'False'} : Bool := FALSE;   // I736.2
      "I736.3" { ExternalVisible := 'False'} : Bool := FALSE;   // I736.3
      "I736.4" { ExternalVisible := 'False'} : Bool := FALSE;   // I736.4
      "I736.5" { ExternalVisible := 'False'} : Bool := FALSE;   // I736.5
      "I736.6" { ExternalVisible := 'False'} : Bool := FALSE;   // I736.6
      "I736.7" { ExternalVisible := 'False'} : Bool := FALSE;   // I736.7
      "I737.0" { ExternalVisible := 'False'} : Bool := FALSE;   // I737.0
      "I737.1" { ExternalVisible := 'False'} : Bool := FALSE;   // I737.1
      "I737.2" { ExternalVisible := 'False'} : Bool := FALSE;   // I737.2
      "I737.3" { ExternalVisible := 'False'} : Bool := FALSE;   // I737.3
      "I737.4" { ExternalVisible := 'False'} : Bool := FALSE;   // I737.4
      "I737.5" { ExternalVisible := 'False'} : Bool := FALSE;   // I737.5
      "I737.6" { ExternalVisible := 'False'} : Bool := FALSE;   // I737.6
      "I737.7" { ExternalVisible := 'False'} : Bool := FALSE;   // I737.7
      "I738.0" { ExternalVisible := 'False'} : Bool := FALSE;   // I738.0
      "I738.1" { ExternalVisible := 'False'} : Bool := FALSE;   // I738.1
      "I738.2" { ExternalVisible := 'False'} : Bool := FALSE;   // I738.2
      "I738.3" { ExternalVisible := 'False'} : Bool := FALSE;   // I738.3
      "I738.4" { ExternalVisible := 'False'} : Bool := FALSE;   // I738.4
      "I738.5" { ExternalVisible := 'False'} : Bool := FALSE;   // I738.5
      "I738.6" { ExternalVisible := 'False'} : Bool := FALSE;   // I738.6
      "I738.7" { ExternalVisible := 'False'} : Bool := FALSE;   // I738.7
      "I739.0" { ExternalVisible := 'False'} : Bool := FALSE;   // I739.0
      "I739.1" { ExternalVisible := 'False'} : Bool := FALSE;   // I739.1
      "I739.2" { ExternalVisible := 'False'} : Bool := FALSE;   // I739.2
      "I739.3" { ExternalVisible := 'False'} : Bool := FALSE;   // I739.3
      "I739.4" { ExternalVisible := 'False'} : Bool := FALSE;   // I739.4
      "I739.5" { ExternalVisible := 'False'} : Bool := FALSE;   // I739.5
      "I739.6" { ExternalVisible := 'False'} : Bool := FALSE;   // I739.6
      "I739.7" { ExternalVisible := 'False'} : Bool := FALSE;   // I739.7
      "I740.0" { ExternalVisible := 'False'} : Bool := FALSE;   // I740.0
      "I740.1" { ExternalVisible := 'False'} : Bool := FALSE;   // I740.1
      "I740.2" { ExternalVisible := 'False'} : Bool := FALSE;   // I740.2
      "I740.3" { ExternalVisible := 'False'} : Bool := FALSE;   // I740.3
      "I740.4" { ExternalVisible := 'False'} : Bool := FALSE;   // I740.4
      "I740.5" { ExternalVisible := 'False'} : Bool := FALSE;   // I740.5
      "I740.6" { ExternalVisible := 'False'} : Bool := FALSE;   // I740.6
      "I740.7" { ExternalVisible := 'False'} : Bool := FALSE;   // I740.7
      "I741.0" { ExternalVisible := 'False'} : Bool := FALSE;   // I741.0
      "I741.1" { ExternalVisible := 'False'} : Bool := FALSE;   // I741.1
      "I741.2" { ExternalVisible := 'False'} : Bool := FALSE;   // I741.2
      "I741.3" { ExternalVisible := 'False'} : Bool := FALSE;   // I741.3
      "I741.4" { ExternalVisible := 'False'} : Bool := FALSE;   // I741.4
      "I741.5" { ExternalVisible := 'False'} : Bool := FALSE;   // I741.5
      "I741.6" { ExternalVisible := 'False'} : Bool := FALSE;   // I741.6
      "I741.7" { ExternalVisible := 'False'} : Bool := FALSE;   // I741.7
      "I742.0" { ExternalVisible := 'False'} : Bool := FALSE;   // I742.0
      "I742.1" { ExternalVisible := 'False'} : Bool := FALSE;   // I742.1
      "I742.2" { ExternalVisible := 'False'} : Bool := FALSE;   // I742.2
      "I742.3" { ExternalVisible := 'False'} : Bool := FALSE;   // I742.3
      "I742.4" { ExternalVisible := 'False'} : Bool := FALSE;   // I742.4
      "I742.5" { ExternalVisible := 'False'} : Bool := FALSE;   // I742.5
      "I742.6" { ExternalVisible := 'False'} : Bool := FALSE;   // I742.6
      "I742.7" { ExternalVisible := 'False'} : Bool := FALSE;   // I742.7
      "I743.0" { ExternalVisible := 'False'} : Bool := FALSE;   // I743.0
      "I743.1" { ExternalVisible := 'False'} : Bool := FALSE;   // I743.1
      "I743.2" { ExternalVisible := 'False'} : Bool := FALSE;   // I743.2
      "I743.3" { ExternalVisible := 'False'} : Bool := FALSE;   // I743.3
      "I743.4" { ExternalVisible := 'False'} : Bool := FALSE;   // I743.4
      "I743.5" { ExternalVisible := 'False'} : Bool := FALSE;   // I743.5
      "I743.6" { ExternalVisible := 'False'} : Bool := FALSE;   // I743.6
      "I743.7" { ExternalVisible := 'False'} : Bool := FALSE;   // I743.7
      "I744.0" { ExternalVisible := 'False'} : Bool := FALSE;   // I744.0
      "I744.1" { ExternalVisible := 'False'} : Bool := FALSE;   // I744.1
      "I744.2" { ExternalVisible := 'False'} : Bool := FALSE;   // I744.2
      "I744.3" { ExternalVisible := 'False'} : Bool := FALSE;   // I744.3
      "I744.4" { ExternalVisible := 'False'} : Bool := FALSE;   // I744.4
      "I744.5" { ExternalVisible := 'False'} : Bool := FALSE;   // I744.5
      "I744.6" { ExternalVisible := 'False'} : Bool := FALSE;   // I744.6
      "I744.7" { ExternalVisible := 'False'} : Bool := FALSE;   // I744.7
      "I745.0" { ExternalVisible := 'False'} : Bool := FALSE;   // I745.0
      "I745.1" { ExternalVisible := 'False'} : Bool := FALSE;   // I745.1
      "I745.2" { ExternalVisible := 'False'} : Bool := FALSE;   // I745.2
      "I745.3" { ExternalVisible := 'False'} : Bool := FALSE;   // I745.3
      "I745.4" { ExternalVisible := 'False'} : Bool := FALSE;   // I745.4
      "I745.5" { ExternalVisible := 'False'} : Bool := FALSE;   // I745.5
      "I745.6" { ExternalVisible := 'False'} : Bool := FALSE;   // I745.6
      "I745.7" { ExternalVisible := 'False'} : Bool := FALSE;   // I745.7
      "I746.0" { ExternalVisible := 'False'} : Bool := FALSE;   // I746.0
      "I746.1" { ExternalVisible := 'False'} : Bool := FALSE;   // I746.1
      "I746.2" { ExternalVisible := 'False'} : Bool := FALSE;   // I746.2
      "I746.3" { ExternalVisible := 'False'} : Bool := FALSE;   // I746.3
      "I746.4" { ExternalVisible := 'False'} : Bool := FALSE;   // I746.4
      "I746.5" { ExternalVisible := 'False'} : Bool := FALSE;   // I746.5
      "I746.6" { ExternalVisible := 'False'} : Bool := FALSE;   // I746.6
      "I746.7" { ExternalVisible := 'False'} : Bool := FALSE;   // I746.7
      "I747.0" { ExternalVisible := 'False'} : Bool := FALSE;   // I747.0
      "I747.1" { ExternalVisible := 'False'} : Bool := FALSE;   // I747.1
      "I747.2" { ExternalVisible := 'False'} : Bool := FALSE;   // I747.2
      "I747.3" { ExternalVisible := 'False'} : Bool := FALSE;   // I747.3
      "I747.4" { ExternalVisible := 'False'} : Bool := FALSE;   // I747.4
      "I747.5" { ExternalVisible := 'False'} : Bool := FALSE;   // I747.5
      "I747.6" { ExternalVisible := 'False'} : Bool := FALSE;   // I747.6
      "I747.7" { ExternalVisible := 'False'} : Bool := FALSE;   // I747.7
      "I748.0" { ExternalVisible := 'False'} : Bool := FALSE;   // I748.0
      "I748.1" { ExternalVisible := 'False'} : Bool := FALSE;   // I748.1
      "I748.2" { ExternalVisible := 'False'} : Bool := FALSE;   // I748.2
      "I748.3" { ExternalVisible := 'False'} : Bool := FALSE;   // I748.3
      "I748.4" { ExternalVisible := 'False'} : Bool := FALSE;   // I748.4
      "I748.5" { ExternalVisible := 'False'} : Bool := FALSE;   // I748.5
      "I748.6" { ExternalVisible := 'False'} : Bool := FALSE;   // I748.6
      "I748.7" { ExternalVisible := 'False'} : Bool := FALSE;   // I748.7
      "I749.0" { ExternalVisible := 'False'} : Bool := FALSE;   // I749.0
      "I749.1" { ExternalVisible := 'False'} : Bool := FALSE;   // I749.1
      "I749.2" { ExternalVisible := 'False'} : Bool := FALSE;   // I749.2
      "I749.3" { ExternalVisible := 'False'} : Bool := FALSE;   // I749.3
      "I749.4" { ExternalVisible := 'False'} : Bool := FALSE;   // I749.4
      "I749.5" { ExternalVisible := 'False'} : Bool := FALSE;   // I749.5
      "I749.6" { ExternalVisible := 'False'} : Bool := FALSE;   // I749.6
      "I749.7" { ExternalVisible := 'False'} : Bool := FALSE;   // I749.7
      "I750.0" { ExternalVisible := 'False'} : Bool := FALSE;   // I750.0
      "I750.1" { ExternalVisible := 'False'} : Bool := FALSE;   // I750.1
      "I750.2" { ExternalVisible := 'False'} : Bool := FALSE;   // I750.2
      "I750.3" { ExternalVisible := 'False'} : Bool := FALSE;   // I750.3
      "I750.4" { ExternalVisible := 'False'} : Bool := FALSE;   // I750.4
      "I750.5" { ExternalVisible := 'False'} : Bool := FALSE;   // I750.5
      "I750.6" { ExternalVisible := 'False'} : Bool := FALSE;   // I750.6
      "I750.7" { ExternalVisible := 'False'} : Bool := FALSE;   // I750.7
      "I751.0" { ExternalVisible := 'False'} : Bool := FALSE;   // I751.0
      "I751.1" { ExternalVisible := 'False'} : Bool := FALSE;   // I751.1
      "I751.2" { ExternalVisible := 'False'} : Bool := FALSE;   // I751.2
      "I751.3" { ExternalVisible := 'False'} : Bool := FALSE;   // I751.3
      "I751.4" { ExternalVisible := 'False'} : Bool := FALSE;   // I751.4
      "I751.5" { ExternalVisible := 'False'} : Bool := FALSE;   // I751.5
      "I751.6" { ExternalVisible := 'False'} : Bool := FALSE;   // I751.6
      "I751.7" { ExternalVisible := 'False'} : Bool := FALSE;   // I751.7
      "I752.0" { ExternalVisible := 'False'} : Bool := FALSE;   // I752.0
      "I752.1" { ExternalVisible := 'False'} : Bool := FALSE;   // I752.1
      "I752.2" { ExternalVisible := 'False'} : Bool := FALSE;   // I752.2
      "I752.3" { ExternalVisible := 'False'} : Bool := FALSE;   // I752.3
      "I752.4" { ExternalVisible := 'False'} : Bool := FALSE;   // I752.4
      "I752.5" { ExternalVisible := 'False'} : Bool := FALSE;   // I752.5
      "I752.6" { ExternalVisible := 'False'} : Bool := FALSE;   // I752.6
      "I752.7" { ExternalVisible := 'False'} : Bool := FALSE;   // I752.7
      "I753.0" { ExternalVisible := 'False'} : Bool := FALSE;   // I753.0
      "I753.1" { ExternalVisible := 'False'} : Bool := FALSE;   // I753.1
      "I753.2" { ExternalVisible := 'False'} : Bool := FALSE;   // I753.2
      "I753.3" { ExternalVisible := 'False'} : Bool := FALSE;   // I753.3
      "I753.4" { ExternalVisible := 'False'} : Bool := FALSE;   // I753.4
      "I753.5" { ExternalVisible := 'False'} : Bool := FALSE;   // I753.5
      "I753.6" { ExternalVisible := 'False'} : Bool := FALSE;   // I753.6
      "I753.7" { ExternalVisible := 'False'} : Bool := FALSE;   // I753.7
      "I754.0" { ExternalVisible := 'False'} : Bool := FALSE;   // I754.0
      "I754.1" { ExternalVisible := 'False'} : Bool := FALSE;   // I754.1
      "I754.2" { ExternalVisible := 'False'} : Bool := FALSE;   // I754.2
      "I754.3" { ExternalVisible := 'False'} : Bool := FALSE;   // I754.3
      "I754.4" { ExternalVisible := 'False'} : Bool := FALSE;   // I754.4
      "I754.5" { ExternalVisible := 'False'} : Bool := FALSE;   // I754.5
      "I754.6" { ExternalVisible := 'False'} : Bool := FALSE;   // I754.6
      "I754.7" { ExternalVisible := 'False'} : Bool := FALSE;   // I754.7
      "I755.0" { ExternalVisible := 'False'} : Bool := FALSE;   // I755.0
      "I755.1" { ExternalVisible := 'False'} : Bool := FALSE;   // I755.1
      "I755.2" { ExternalVisible := 'False'} : Bool := FALSE;   // I755.2
      "I755.3" { ExternalVisible := 'False'} : Bool := FALSE;   // I755.3
      "I755.4" { ExternalVisible := 'False'} : Bool := FALSE;   // I755.4
      "I755.5" { ExternalVisible := 'False'} : Bool := FALSE;   // I755.5
      "I755.6" { ExternalVisible := 'False'} : Bool := FALSE;   // I755.6
      "I755.7" { ExternalVisible := 'False'} : Bool := FALSE;   // I755.7
      "I756.0" { ExternalVisible := 'False'} : Bool := FALSE;   // I756.0
      "I756.1" { ExternalVisible := 'False'} : Bool := FALSE;   // I756.1
      "I756.2" { ExternalVisible := 'False'} : Bool := FALSE;   // I756.2
      "I756.3" { ExternalVisible := 'False'} : Bool := FALSE;   // I756.3
      "I756.4" { ExternalVisible := 'False'} : Bool := FALSE;   // I756.4
      "I756.5" { ExternalVisible := 'False'} : Bool := FALSE;   // I756.5
      "I756.6" { ExternalVisible := 'False'} : Bool := FALSE;   // I756.6
      "I756.7" { ExternalVisible := 'False'} : Bool := FALSE;   // I756.7
      "I757.0" { ExternalVisible := 'False'} : Bool := FALSE;   // I757.0
      "I757.1" { ExternalVisible := 'False'} : Bool := FALSE;   // I757.1
      "I757.2" { ExternalVisible := 'False'} : Bool := FALSE;   // I757.2
      "I757.3" { ExternalVisible := 'False'} : Bool := FALSE;   // I757.3
      "I757.4" { ExternalVisible := 'False'} : Bool := FALSE;   // I757.4
      "I757.5" { ExternalVisible := 'False'} : Bool := FALSE;   // I757.5
      "I757.6" { ExternalVisible := 'False'} : Bool := FALSE;   // I757.6
      "I757.7" { ExternalVisible := 'False'} : Bool := FALSE;   // I757.7
      "I758.0" { ExternalVisible := 'False'} : Bool := FALSE;   // I758.0
      "I758.1" { ExternalVisible := 'False'} : Bool := FALSE;   // I758.1
      "I758.2" { ExternalVisible := 'False'} : Bool := FALSE;   // I758.2
      "I758.3" { ExternalVisible := 'False'} : Bool := FALSE;   // I758.3
      "I758.4" { ExternalVisible := 'False'} : Bool := FALSE;   // I758.4
      "I758.5" { ExternalVisible := 'False'} : Bool := FALSE;   // I758.5
      "I758.6" { ExternalVisible := 'False'} : Bool := FALSE;   // I758.6
      "I758.7" { ExternalVisible := 'False'} : Bool := FALSE;   // I758.7
      "I759.0" { ExternalVisible := 'False'} : Bool := FALSE;   // I759.0
      "I759.1" { ExternalVisible := 'False'} : Bool := FALSE;   // I759.1
      "I759.2" { ExternalVisible := 'False'} : Bool := FALSE;   // I759.2
      "I759.3" { ExternalVisible := 'False'} : Bool := FALSE;   // I759.3
      "I759.4" { ExternalVisible := 'False'} : Bool := FALSE;   // I759.4
      "I759.5" { ExternalVisible := 'False'} : Bool := FALSE;   // I759.5
      "I759.6" { ExternalVisible := 'False'} : Bool := FALSE;   // I759.6
      "I759.7" { ExternalVisible := 'False'} : Bool := FALSE;   // I759.7
      "I760.0" { ExternalVisible := 'False'} : Bool := FALSE;   // I760.0
      "I760.1" { ExternalVisible := 'False'} : Bool := FALSE;   // I760.1
      "I760.2" { ExternalVisible := 'False'} : Bool := FALSE;   // I760.2
      "I760.3" { ExternalVisible := 'False'} : Bool := FALSE;   // I760.3
      "I760.4" { ExternalVisible := 'False'} : Bool := FALSE;   // I760.4
      "I760.5" { ExternalVisible := 'False'} : Bool := FALSE;   // I760.5
      "I760.6" { ExternalVisible := 'False'} : Bool := FALSE;   // I760.6
      "I760.7" { ExternalVisible := 'False'} : Bool := FALSE;   // I760.7
      "I761.0" { ExternalVisible := 'False'} : Bool := FALSE;   // I761.0
      "I761.1" { ExternalVisible := 'False'} : Bool := FALSE;   // I761.1
      "I761.2" { ExternalVisible := 'False'} : Bool := FALSE;   // I761.2
      "I761.3" { ExternalVisible := 'False'} : Bool := FALSE;   // I761.3
      "I761.4" { ExternalVisible := 'False'} : Bool := FALSE;   // I761.4
      "I761.5" { ExternalVisible := 'False'} : Bool := FALSE;   // I761.5
      "I761.6" { ExternalVisible := 'False'} : Bool := FALSE;   // I761.6
      "I761.7" { ExternalVisible := 'False'} : Bool := FALSE;   // I761.7
      "I762.0" { ExternalVisible := 'False'} : Bool := FALSE;   // I762.0
      "I762.1" { ExternalVisible := 'False'} : Bool := FALSE;   // I762.1
      "I762.2" { ExternalVisible := 'False'} : Bool := FALSE;   // I762.2
      "I762.3" { ExternalVisible := 'False'} : Bool := FALSE;   // I762.3
      "I762.4" { ExternalVisible := 'False'} : Bool := FALSE;   // I762.4
      "I762.5" { ExternalVisible := 'False'} : Bool := FALSE;   // I762.5
      "I762.6" { ExternalVisible := 'False'} : Bool := FALSE;   // I762.6
      "I762.7" { ExternalVisible := 'False'} : Bool := FALSE;   // I762.7
      "I763.0" { ExternalVisible := 'False'} : Bool := FALSE;   // I763.0
      "I763.1" { ExternalVisible := 'False'} : Bool := FALSE;   // I763.1
      "I763.2" { ExternalVisible := 'False'} : Bool := FALSE;   // I763.2
      "I763.3" { ExternalVisible := 'False'} : Bool := FALSE;   // I763.3
      "I763.4" { ExternalVisible := 'False'} : Bool := FALSE;   // I763.4
      "I763.5" { ExternalVisible := 'False'} : Bool := FALSE;   // I763.5
      "I763.6" { ExternalVisible := 'False'} : Bool := FALSE;   // I763.6
      "I763.7" { ExternalVisible := 'False'} : Bool := FALSE;   // I763.7
      "I764.0" { ExternalVisible := 'False'} : Bool := FALSE;   // I764.0
      "I764.1" { ExternalVisible := 'False'} : Bool := FALSE;   // I764.1
      "I764.2" { ExternalVisible := 'False'} : Bool := FALSE;   // I764.2
      "I764.3" { ExternalVisible := 'False'} : Bool := FALSE;   // I764.3
      "I764.4" { ExternalVisible := 'False'} : Bool := FALSE;   // I764.4
      "I764.5" { ExternalVisible := 'False'} : Bool := FALSE;   // I764.5
      "I764.6" { ExternalVisible := 'False'} : Bool := FALSE;   // I764.6
      "I764.7" { ExternalVisible := 'False'} : Bool := FALSE;   // I764.7
      "I765.0" { ExternalVisible := 'False'} : Bool := FALSE;   // I765.0
      "I765.1" { ExternalVisible := 'False'} : Bool := FALSE;   // I765.1
      "I765.2" { ExternalVisible := 'False'} : Bool := FALSE;   // I765.2
      "I765.3" { ExternalVisible := 'False'} : Bool := FALSE;   // I765.3
      "I765.4" { ExternalVisible := 'False'} : Bool := FALSE;   // I765.4
      "I765.5" { ExternalVisible := 'False'} : Bool := FALSE;   // I765.5
      "I765.6" { ExternalVisible := 'False'} : Bool := FALSE;   // I765.6
      "I765.7" { ExternalVisible := 'False'} : Bool := FALSE;   // I765.7
      "I766.0" { ExternalVisible := 'False'} : Bool := FALSE;   // I766.0
      "I766.1" { ExternalVisible := 'False'} : Bool := FALSE;   // I766.1
      "I766.2" { ExternalVisible := 'False'} : Bool := FALSE;   // I766.2
      "I766.3" { ExternalVisible := 'False'} : Bool := FALSE;   // I766.3
      "I766.4" { ExternalVisible := 'False'} : Bool := FALSE;   // I766.4
      "I766.5" { ExternalVisible := 'False'} : Bool := FALSE;   // I766.5
      "I766.6" { ExternalVisible := 'False'} : Bool := FALSE;   // I766.6
      "I766.7" { ExternalVisible := 'False'} : Bool := FALSE;   // I766.7
      "I767.0" { ExternalVisible := 'False'} : Bool := FALSE;   // I767.0
      "I767.1" { ExternalVisible := 'False'} : Bool := FALSE;   // I767.1
      "I767.2" { ExternalVisible := 'False'} : Bool := FALSE;   // I767.2
      "I767.3" { ExternalVisible := 'False'} : Bool := FALSE;   // I767.3
      "I767.4" { ExternalVisible := 'False'} : Bool := FALSE;   // I767.4
      "I767.5" { ExternalVisible := 'False'} : Bool := FALSE;   // I767.5
      "I767.6" { ExternalVisible := 'False'} : Bool := FALSE;   // I767.6
      "I767.7" { ExternalVisible := 'False'} : Bool := FALSE;   // I767.7
      "I768.0" { ExternalVisible := 'False'} : Bool := FALSE;   // I768.0
      "I768.1" { ExternalVisible := 'False'} : Bool := FALSE;   // I768.1
      "I768.2" { ExternalVisible := 'False'} : Bool := FALSE;   // I768.2
      "I768.3" { ExternalVisible := 'False'} : Bool := FALSE;   // I768.3
      "I768.4" { ExternalVisible := 'False'} : Bool := FALSE;   // I768.4
      "I768.5" { ExternalVisible := 'False'} : Bool := FALSE;   // I768.5
      "I768.6" { ExternalVisible := 'False'} : Bool := FALSE;   // I768.6
      "I768.7" { ExternalVisible := 'False'} : Bool := FALSE;   // I768.7
      "I769.0" { ExternalVisible := 'False'} : Bool := FALSE;   // I769.0
      "I769.1" { ExternalVisible := 'False'} : Bool := FALSE;   // I769.1
      "I769.2" { ExternalVisible := 'False'} : Bool := FALSE;   // I769.2
      "I769.3" { ExternalVisible := 'False'} : Bool := FALSE;   // I769.3
      "I769.4" { ExternalVisible := 'False'} : Bool := FALSE;   // I769.4
      "I769.5" { ExternalVisible := 'False'} : Bool := FALSE;   // I769.5
      "I769.6" { ExternalVisible := 'False'} : Bool := FALSE;   // I769.6
      "I769.7" { ExternalVisible := 'False'} : Bool := FALSE;   // I769.7
      "I770.0" { ExternalVisible := 'False'} : Bool := FALSE;   // I770.0
      "I770.1" { ExternalVisible := 'False'} : Bool := FALSE;   // I770.1
      "I770.2" { ExternalVisible := 'False'} : Bool := FALSE;   // I770.2
      "I770.3" { ExternalVisible := 'False'} : Bool := FALSE;   // I770.3
      "I770.4" { ExternalVisible := 'False'} : Bool := FALSE;   // I770.4
      "I770.5" { ExternalVisible := 'False'} : Bool := FALSE;   // I770.5
      "I770.6" { ExternalVisible := 'False'} : Bool := FALSE;   // I770.6
      "I770.7" { ExternalVisible := 'False'} : Bool := FALSE;   // I770.7
      "I771.0" { ExternalVisible := 'False'} : Bool := FALSE;   // I771.0
      "I771.1" { ExternalVisible := 'False'} : Bool := FALSE;   // I771.1
      "I771.2" { ExternalVisible := 'False'} : Bool := FALSE;   // I771.2
      "I771.3" { ExternalVisible := 'False'} : Bool := FALSE;   // I771.3
      "I771.4" { ExternalVisible := 'False'} : Bool := FALSE;   // I771.4
      "I771.5" { ExternalVisible := 'False'} : Bool := FALSE;   // I771.5
      "I771.6" { ExternalVisible := 'False'} : Bool := FALSE;   // I771.6
      "I771.7" { ExternalVisible := 'False'} : Bool := FALSE;   // I771.7
      "I772.0" { ExternalVisible := 'False'} : Bool := FALSE;   // I772.0
      "I772.1" { ExternalVisible := 'False'} : Bool := FALSE;   // I772.1
      "I772.2" { ExternalVisible := 'False'} : Bool := FALSE;   // I772.2
      "I772.3" { ExternalVisible := 'False'} : Bool := FALSE;   // I772.3
      "I772.4" { ExternalVisible := 'False'} : Bool := FALSE;   // I772.4
      "I772.5" { ExternalVisible := 'False'} : Bool := FALSE;   // I772.5
      "I772.6" { ExternalVisible := 'False'} : Bool := FALSE;   // I772.6
      "I772.7" { ExternalVisible := 'False'} : Bool := FALSE;   // I772.7
      "I773.0" { ExternalVisible := 'False'} : Bool := FALSE;   // I773.0
      "I773.1" { ExternalVisible := 'False'} : Bool := FALSE;   // I773.1
      "I773.2" { ExternalVisible := 'False'} : Bool := FALSE;   // I773.2
      "I773.3" { ExternalVisible := 'False'} : Bool := FALSE;   // I773.3
      "I773.4" { ExternalVisible := 'False'} : Bool := FALSE;   // I773.4
      "I773.5" { ExternalVisible := 'False'} : Bool := FALSE;   // I773.5
      "I773.6" { ExternalVisible := 'False'} : Bool := FALSE;   // I773.6
      "I773.7" { ExternalVisible := 'False'} : Bool := FALSE;   // I773.7
      "I774.0" { ExternalVisible := 'False'} : Bool := FALSE;   // I774.0
      "I774.1" { ExternalVisible := 'False'} : Bool := FALSE;   // I774.1
      "I774.2" { ExternalVisible := 'False'} : Bool := FALSE;   // I774.2
      "I774.3" { ExternalVisible := 'False'} : Bool := FALSE;   // I774.3
      "I774.4" { ExternalVisible := 'False'} : Bool := FALSE;   // I774.4
      "I774.5" { ExternalVisible := 'False'} : Bool := FALSE;   // I774.5
      "I774.6" { ExternalVisible := 'False'} : Bool := FALSE;   // I774.6
      "I774.7" { ExternalVisible := 'False'} : Bool := FALSE;   // I774.7
      "I775.0" { ExternalVisible := 'False'} : Bool := FALSE;   // I775.0
      "I775.1" { ExternalVisible := 'False'} : Bool := FALSE;   // I775.1
      "I775.2" { ExternalVisible := 'False'} : Bool := FALSE;   // I775.2
      "I775.3" { ExternalVisible := 'False'} : Bool := FALSE;   // I775.3
      "I775.4" { ExternalVisible := 'False'} : Bool := FALSE;   // I775.4
      "I775.5" { ExternalVisible := 'False'} : Bool := FALSE;   // I775.5
      "I775.6" { ExternalVisible := 'False'} : Bool := FALSE;   // I775.6
      "I775.7" { ExternalVisible := 'False'} : Bool := FALSE;   // I775.7
      "I776.0" { ExternalVisible := 'False'} : Bool := FALSE;   // I776.0
      "I776.1" { ExternalVisible := 'False'} : Bool := FALSE;   // I776.1
      "I776.2" { ExternalVisible := 'False'} : Bool := FALSE;   // I776.2
      "I776.3" { ExternalVisible := 'False'} : Bool := FALSE;   // I776.3
      "I776.4" { ExternalVisible := 'False'} : Bool := FALSE;   // I776.4
      "I776.5" { ExternalVisible := 'False'} : Bool := FALSE;   // I776.5
      "I776.6" { ExternalVisible := 'False'} : Bool := FALSE;   // I776.6
      "I776.7" { ExternalVisible := 'False'} : Bool := FALSE;   // I776.7
      "I777.0" { ExternalVisible := 'False'} : Bool := FALSE;   // I777.0
      "I777.1" { ExternalVisible := 'False'} : Bool := FALSE;   // I777.1
      "I777.2" { ExternalVisible := 'False'} : Bool := FALSE;   // I777.2
      "I777.3" { ExternalVisible := 'False'} : Bool := FALSE;   // I777.3
      "I777.4" { ExternalVisible := 'False'} : Bool := FALSE;   // I777.4
      "I777.5" { ExternalVisible := 'False'} : Bool := FALSE;   // I777.5
      "I777.6" { ExternalVisible := 'False'} : Bool := FALSE;   // I777.6
      "I777.7" { ExternalVisible := 'False'} : Bool := FALSE;   // I777.7
      "I778.0" { ExternalVisible := 'False'} : Bool := FALSE;   // I778.0
      "I778.1" { ExternalVisible := 'False'} : Bool := FALSE;   // I778.1
      "I778.2" { ExternalVisible := 'False'} : Bool := FALSE;   // I778.2
      "I778.3" { ExternalVisible := 'False'} : Bool := FALSE;   // I778.3
      "I778.4" { ExternalVisible := 'False'} : Bool := FALSE;   // I778.4
      "I778.5" { ExternalVisible := 'False'} : Bool := FALSE;   // I778.5
      "I778.6" { ExternalVisible := 'False'} : Bool := FALSE;   // I778.6
      "I778.7" { ExternalVisible := 'False'} : Bool := FALSE;   // I778.7
      "I779.0" { ExternalVisible := 'False'} : Bool := FALSE;   // I779.0
      "I779.1" { ExternalVisible := 'False'} : Bool := FALSE;   // I779.1
      "I779.2" { ExternalVisible := 'False'} : Bool := FALSE;   // I779.2
      "I779.3" { ExternalVisible := 'False'} : Bool := FALSE;   // I779.3
      "I779.4" { ExternalVisible := 'False'} : Bool := FALSE;   // I779.4
      "I779.5" { ExternalVisible := 'False'} : Bool := FALSE;   // I779.5
      "I779.6" { ExternalVisible := 'False'} : Bool := FALSE;   // I779.6
      "I779.7" { ExternalVisible := 'False'} : Bool := FALSE;   // I779.7
      "I780.0" { ExternalVisible := 'False'} : Bool := FALSE;   // I780.0
      "I780.1" { ExternalVisible := 'False'} : Bool := FALSE;   // I780.1
      "I780.2" { ExternalVisible := 'False'} : Bool := FALSE;   // I780.2
      "I780.3" { ExternalVisible := 'False'} : Bool := FALSE;   // I780.3
      "I780.4" { ExternalVisible := 'False'} : Bool := FALSE;   // I780.4
      "I780.5" { ExternalVisible := 'False'} : Bool := FALSE;   // I780.5
      "I780.6" { ExternalVisible := 'False'} : Bool := FALSE;   // I780.6
      "I780.7" { ExternalVisible := 'False'} : Bool := FALSE;   // I780.7
      "I781.0" { ExternalVisible := 'False'} : Bool := FALSE;   // I781.0
      "I781.1" { ExternalVisible := 'False'} : Bool := FALSE;   // I781.1
      "I781.2" { ExternalVisible := 'False'} : Bool := FALSE;   // I781.2
      "I781.3" { ExternalVisible := 'False'} : Bool := FALSE;   // I781.3
      "I781.4" { ExternalVisible := 'False'} : Bool := FALSE;   // I781.4
      "I781.5" { ExternalVisible := 'False'} : Bool := FALSE;   // I781.5
      "I781.6" { ExternalVisible := 'False'} : Bool := FALSE;   // I781.6
      "I781.7" { ExternalVisible := 'False'} : Bool := FALSE;   // I781.7
      "I782.0" { ExternalVisible := 'False'} : Bool := FALSE;   // I782.0
      "I782.1" { ExternalVisible := 'False'} : Bool := FALSE;   // I782.1
      "I782.2" { ExternalVisible := 'False'} : Bool := FALSE;   // I782.2
      "I782.3" { ExternalVisible := 'False'} : Bool := FALSE;   // I782.3
      "I782.4" { ExternalVisible := 'False'} : Bool := FALSE;   // I782.4
      "I782.5" { ExternalVisible := 'False'} : Bool := FALSE;   // I782.5
      "I782.6" { ExternalVisible := 'False'} : Bool := FALSE;   // I782.6
      "I782.7" { ExternalVisible := 'False'} : Bool := FALSE;   // I782.7
      "I783.0" { ExternalVisible := 'False'} : Bool := FALSE;   // I783.0
      "I783.1" { ExternalVisible := 'False'} : Bool := FALSE;   // I783.1
      "I783.2" { ExternalVisible := 'False'} : Bool := FALSE;   // I783.2
      "I783.3" { ExternalVisible := 'False'} : Bool := FALSE;   // I783.3
      "I783.4" { ExternalVisible := 'False'} : Bool := FALSE;   // I783.4
      "I783.5" { ExternalVisible := 'False'} : Bool := FALSE;   // I783.5
      "I783.6" { ExternalVisible := 'False'} : Bool := FALSE;   // I783.6
      "I783.7" { ExternalVisible := 'False'} : Bool := FALSE;   // I783.7
      "I784.0" { ExternalVisible := 'False'} : Bool := FALSE;   // I784.0
      "I784.1" { ExternalVisible := 'False'} : Bool := FALSE;   // I784.1
      "I784.2" { ExternalVisible := 'False'} : Bool := FALSE;   // I784.2
      "I784.3" { ExternalVisible := 'False'} : Bool := FALSE;   // I784.3
      "I784.4" { ExternalVisible := 'False'} : Bool := FALSE;   // I784.4
      "I784.5" { ExternalVisible := 'False'} : Bool := FALSE;   // I784.5
      "I784.6" { ExternalVisible := 'False'} : Bool := FALSE;   // I784.6
      "I784.7" { ExternalVisible := 'False'} : Bool := FALSE;   // I784.7
      "I785.0" { ExternalVisible := 'False'} : Bool := FALSE;   // I785.0
      "I785.1" { ExternalVisible := 'False'} : Bool := FALSE;   // I785.1
      "I785.2" { ExternalVisible := 'False'} : Bool := FALSE;   // I785.2
      "I785.3" { ExternalVisible := 'False'} : Bool := FALSE;   // I785.3
      "I785.4" { ExternalVisible := 'False'} : Bool := FALSE;   // I785.4
      "I785.5" { ExternalVisible := 'False'} : Bool := FALSE;   // I785.5
      "I785.6" { ExternalVisible := 'False'} : Bool := FALSE;   // I785.6
      "I785.7" { ExternalVisible := 'False'} : Bool := FALSE;   // I785.7
      "I786.0" { ExternalVisible := 'False'} : Bool := FALSE;   // I786.0
      "I786.1" { ExternalVisible := 'False'} : Bool := FALSE;   // I786.1
      "I786.2" { ExternalVisible := 'False'} : Bool := FALSE;   // I786.2
      "I786.3" { ExternalVisible := 'False'} : Bool := FALSE;   // I786.3
      "I786.4" { ExternalVisible := 'False'} : Bool := FALSE;   // I786.4
      "I786.5" { ExternalVisible := 'False'} : Bool := FALSE;   // I786.5
      "I786.6" { ExternalVisible := 'False'} : Bool := FALSE;   // I786.6
      "I786.7" { ExternalVisible := 'False'} : Bool := FALSE;   // I786.7
      "I787.0" { ExternalVisible := 'False'} : Bool := FALSE;   // I787.0
      "I787.1" { ExternalVisible := 'False'} : Bool := FALSE;   // I787.1
      "I787.2" { ExternalVisible := 'False'} : Bool := FALSE;   // I787.2
      "I787.3" { ExternalVisible := 'False'} : Bool := FALSE;   // I787.3
      "I787.4" { ExternalVisible := 'False'} : Bool := FALSE;   // I787.4
      "I787.5" { ExternalVisible := 'False'} : Bool := FALSE;   // I787.5
      "I787.6" { ExternalVisible := 'False'} : Bool := FALSE;   // I787.6
      "I787.7" { ExternalVisible := 'False'} : Bool := FALSE;   // I787.7
      "I788.0" { ExternalVisible := 'False'} : Bool := FALSE;   // I788.0
      "I788.1" { ExternalVisible := 'False'} : Bool := FALSE;   // I788.1
      "I788.2" { ExternalVisible := 'False'} : Bool := FALSE;   // I788.2
      "I788.3" { ExternalVisible := 'False'} : Bool := FALSE;   // I788.3
      "I788.4" { ExternalVisible := 'False'} : Bool := FALSE;   // I788.4
      "I788.5" { ExternalVisible := 'False'} : Bool := FALSE;   // I788.5
      "I788.6" { ExternalVisible := 'False'} : Bool := FALSE;   // I788.6
      "I788.7" { ExternalVisible := 'False'} : Bool := FALSE;   // I788.7
      "I789.0" { ExternalVisible := 'False'} : Bool := FALSE;   // I789.0
      "I789.1" { ExternalVisible := 'False'} : Bool := FALSE;   // I789.1
      "I789.2" { ExternalVisible := 'False'} : Bool := FALSE;   // I789.2
      "I789.3" { ExternalVisible := 'False'} : Bool := FALSE;   // I789.3
      "I789.4" { ExternalVisible := 'False'} : Bool := FALSE;   // I789.4
      "I789.5" { ExternalVisible := 'False'} : Bool := FALSE;   // I789.5
      "I789.6" { ExternalVisible := 'False'} : Bool := FALSE;   // I789.6
      "I789.7" { ExternalVisible := 'False'} : Bool := FALSE;   // I789.7
      "I790.0" { ExternalVisible := 'False'} : Bool := FALSE;   // I790.0
      "I790.1" { ExternalVisible := 'False'} : Bool := FALSE;   // I790.1
      "I790.2" { ExternalVisible := 'False'} : Bool := FALSE;   // I790.2
      "I790.3" { ExternalVisible := 'False'} : Bool := FALSE;   // I790.3
      "I790.4" { ExternalVisible := 'False'} : Bool := FALSE;   // I790.4
      "I790.5" { ExternalVisible := 'False'} : Bool := FALSE;   // I790.5
      "I790.6" { ExternalVisible := 'False'} : Bool := FALSE;   // I790.6
      "I790.7" { ExternalVisible := 'False'} : Bool := FALSE;   // I790.7
      "I791.0" { ExternalVisible := 'False'} : Bool := FALSE;   // I791.0
      "I791.1" { ExternalVisible := 'False'} : Bool := FALSE;   // I791.1
      "I791.2" { ExternalVisible := 'False'} : Bool := FALSE;   // I791.2
      "I791.3" { ExternalVisible := 'False'} : Bool := FALSE;   // I791.3
      "I791.4" { ExternalVisible := 'False'} : Bool := FALSE;   // I791.4
      "I791.5" { ExternalVisible := 'False'} : Bool := FALSE;   // I791.5
      "I791.6" { ExternalVisible := 'False'} : Bool := FALSE;   // I791.6
      "I791.7" { ExternalVisible := 'False'} : Bool := FALSE;   // I791.7
      "I792.0" { ExternalVisible := 'False'} : Bool := FALSE;   // I792.0
      "I792.1" { ExternalVisible := 'False'} : Bool := FALSE;   // I792.1
      "I792.2" { ExternalVisible := 'False'} : Bool := FALSE;   // I792.2
      "I792.3" { ExternalVisible := 'False'} : Bool := FALSE;   // I792.3
      "I792.4" { ExternalVisible := 'False'} : Bool := FALSE;   // I792.4
      "I792.5" { ExternalVisible := 'False'} : Bool := FALSE;   // I792.5
      "I792.6" { ExternalVisible := 'False'} : Bool := FALSE;   // I792.6
      "I792.7" { ExternalVisible := 'False'} : Bool := FALSE;   // I792.7
      "I793.0" { ExternalVisible := 'False'} : Bool := FALSE;   // I793.0
      "I793.1" { ExternalVisible := 'False'} : Bool := FALSE;   // I793.1
      "I793.2" { ExternalVisible := 'False'} : Bool := FALSE;   // I793.2
      "I793.3" { ExternalVisible := 'False'} : Bool := FALSE;   // I793.3
      "I793.4" { ExternalVisible := 'False'} : Bool := FALSE;   // I793.4
      "I793.5" { ExternalVisible := 'False'} : Bool := FALSE;   // I793.5
      "I793.6" { ExternalVisible := 'False'} : Bool := FALSE;   // I793.6
      "I793.7" { ExternalVisible := 'False'} : Bool := FALSE;   // I793.7
      "I794.0" { ExternalVisible := 'False'} : Bool := FALSE;   // I794.0
      "I794.1" { ExternalVisible := 'False'} : Bool := FALSE;   // I794.1
      "I794.2" { ExternalVisible := 'False'} : Bool := FALSE;   // I794.2
      "I794.3" { ExternalVisible := 'False'} : Bool := FALSE;   // I794.3
      "I794.4" { ExternalVisible := 'False'} : Bool := FALSE;   // I794.4
      "I794.5" { ExternalVisible := 'False'} : Bool := FALSE;   // I794.5
      "I794.6" { ExternalVisible := 'False'} : Bool := FALSE;   // I794.6
      "I794.7" { ExternalVisible := 'False'} : Bool := FALSE;   // I794.7
      "I795.0" { ExternalVisible := 'False'} : Bool := FALSE;   // I795.0
      "I795.1" { ExternalVisible := 'False'} : Bool := FALSE;   // I795.1
      "I795.2" { ExternalVisible := 'False'} : Bool := FALSE;   // I795.2
      "I795.3" { ExternalVisible := 'False'} : Bool := FALSE;   // I795.3
      "I795.4" { ExternalVisible := 'False'} : Bool := FALSE;   // I795.4
      "I795.5" { ExternalVisible := 'False'} : Bool := FALSE;   // I795.5
      "I795.6" { ExternalVisible := 'False'} : Bool := FALSE;   // I795.6
      "I795.7" { ExternalVisible := 'False'} : Bool := FALSE;   // I795.7
      "I796.0" { ExternalVisible := 'False'} : Bool := FALSE;   // I796.0
      "I796.1" { ExternalVisible := 'False'} : Bool := FALSE;   // I796.1
      "I796.2" { ExternalVisible := 'False'} : Bool := FALSE;   // I796.2
      "I796.3" { ExternalVisible := 'False'} : Bool := FALSE;   // I796.3
      "I796.4" { ExternalVisible := 'False'} : Bool := FALSE;   // I796.4
      "I796.5" { ExternalVisible := 'False'} : Bool := FALSE;   // I796.5
      "I796.6" { ExternalVisible := 'False'} : Bool := FALSE;   // I796.6
      "I796.7" { ExternalVisible := 'False'} : Bool := FALSE;   // I796.7
      "I797.0" { ExternalVisible := 'False'} : Bool := FALSE;   // I797.0
      "I797.1" { ExternalVisible := 'False'} : Bool := FALSE;   // I797.1
      "I797.2" { ExternalVisible := 'False'} : Bool := FALSE;   // I797.2
      "I797.3" { ExternalVisible := 'False'} : Bool := FALSE;   // I797.3
      "I797.4" { ExternalVisible := 'False'} : Bool := FALSE;   // I797.4
      "I797.5" { ExternalVisible := 'False'} : Bool := FALSE;   // I797.5
      "I797.6" { ExternalVisible := 'False'} : Bool := FALSE;   // I797.6
      "I797.7" { ExternalVisible := 'False'} : Bool := FALSE;   // I797.7
      "I798.0" { ExternalVisible := 'False'} : Bool := FALSE;   // I798.0
      "I798.1" { ExternalVisible := 'False'} : Bool := FALSE;   // I798.1
      "I798.2" { ExternalVisible := 'False'} : Bool := FALSE;   // I798.2
      "I798.3" { ExternalVisible := 'False'} : Bool := FALSE;   // I798.3
      "I798.4" { ExternalVisible := 'False'} : Bool := FALSE;   // I798.4
      "I798.5" { ExternalVisible := 'False'} : Bool := FALSE;   // I798.5
      "I798.6" { ExternalVisible := 'False'} : Bool := FALSE;   // I798.6
      "I798.7" { ExternalVisible := 'False'} : Bool := FALSE;   // I798.7
      "I799.0" { ExternalVisible := 'False'} : Bool := FALSE;   // I799.0
      "I799.1" { ExternalVisible := 'False'} : Bool := FALSE;   // I799.1
      "I799.2" { ExternalVisible := 'False'} : Bool := FALSE;   // I799.2
      "I799.3" { ExternalVisible := 'False'} : Bool := FALSE;   // I799.3
      "I799.4" { ExternalVisible := 'False'} : Bool := FALSE;   // I799.4
      "I799.5" { ExternalVisible := 'False'} : Bool := FALSE;   // I799.5
      "I799.6" { ExternalVisible := 'False'} : Bool := FALSE;   // I799.6
      "I799.7" { ExternalVisible := 'False'} : Bool := FALSE;   // I799.7
      "I800.0" { ExternalVisible := 'False'} : Bool := FALSE;   // I800.0
      "I800.1" { ExternalVisible := 'False'} : Bool := FALSE;   // I800.1
      "I800.2" { ExternalVisible := 'False'} : Bool := FALSE;   // I800.2
      "I800.3" { ExternalVisible := 'False'} : Bool := FALSE;   // I800.3
      "I800.4" { ExternalVisible := 'False'} : Bool := FALSE;   // I800.4
      "I800.5" { ExternalVisible := 'False'} : Bool := FALSE;   // I800.5
      "I800.6" { ExternalVisible := 'False'} : Bool := FALSE;   // I800.6
      "I800.7" { ExternalVisible := 'False'} : Bool := FALSE;   // I800.7
      "I801.0" { ExternalVisible := 'False'} : Bool := FALSE;   // I801.0
      "I801.1" { ExternalVisible := 'False'} : Bool := FALSE;   // I801.1
      "I801.2" { ExternalVisible := 'False'} : Bool := FALSE;   // I801.2
      "I801.3" { ExternalVisible := 'False'} : Bool := FALSE;   // I801.3
      "I801.4" { ExternalVisible := 'False'} : Bool := FALSE;   // I801.4
      "I801.5" { ExternalVisible := 'False'} : Bool := FALSE;   // I801.5
      "I801.6" { ExternalVisible := 'False'} : Bool := FALSE;   // I801.6
      "I801.7" { ExternalVisible := 'False'} : Bool := FALSE;   // I801.7
      "I802.0" { ExternalVisible := 'False'} : Bool := FALSE;   // I802.0
      "I802.1" { ExternalVisible := 'False'} : Bool := FALSE;   // I802.1
      "I802.2" { ExternalVisible := 'False'} : Bool := FALSE;   // I802.2
      "I802.3" { ExternalVisible := 'False'} : Bool := FALSE;   // I802.3
      "I802.4" { ExternalVisible := 'False'} : Bool := FALSE;   // I802.4
      "I802.5" { ExternalVisible := 'False'} : Bool := FALSE;   // I802.5
      "I802.6" { ExternalVisible := 'False'} : Bool := FALSE;   // I802.6
      "I802.7" { ExternalVisible := 'False'} : Bool := FALSE;   // I802.7
      "I803.0" { ExternalVisible := 'False'} : Bool := FALSE;   // I803.0
      "I803.1" { ExternalVisible := 'False'} : Bool := FALSE;   // I803.1
      "I803.2" { ExternalVisible := 'False'} : Bool := FALSE;   // I803.2
      "I803.3" { ExternalVisible := 'False'} : Bool := FALSE;   // I803.3
      "I803.4" { ExternalVisible := 'False'} : Bool := FALSE;   // I803.4
      "I803.5" { ExternalVisible := 'False'} : Bool := FALSE;   // I803.5
      "I803.6" { ExternalVisible := 'False'} : Bool := FALSE;   // I803.6
      "I803.7" { ExternalVisible := 'False'} : Bool := FALSE;   // I803.7
      "I804.0" { ExternalVisible := 'False'} : Bool := FALSE;   // I804.0
      "I804.1" { ExternalVisible := 'False'} : Bool := FALSE;   // I804.1
      "I804.2" { ExternalVisible := 'False'} : Bool := FALSE;   // I804.2
      "I804.3" { ExternalVisible := 'False'} : Bool := FALSE;   // I804.3
      "I804.4" { ExternalVisible := 'False'} : Bool := FALSE;   // I804.4
      "I804.5" { ExternalVisible := 'False'} : Bool := FALSE;   // I804.5
      "I804.6" { ExternalVisible := 'False'} : Bool := FALSE;   // I804.6
      "I804.7" { ExternalVisible := 'False'} : Bool := FALSE;   // I804.7
      "I805.0" { ExternalVisible := 'False'} : Bool := FALSE;   // I805.0
      "I805.1" { ExternalVisible := 'False'} : Bool := FALSE;   // I805.1
      "I805.2" { ExternalVisible := 'False'} : Bool := FALSE;   // I805.2
      "I805.3" { ExternalVisible := 'False'} : Bool := FALSE;   // I805.3
      "I805.4" { ExternalVisible := 'False'} : Bool := FALSE;   // I805.4
      "I805.5" { ExternalVisible := 'False'} : Bool := FALSE;   // I805.5
      "I805.6" { ExternalVisible := 'False'} : Bool := FALSE;   // I805.6
      "I805.7" { ExternalVisible := 'False'} : Bool := FALSE;   // I805.7
      "I806.0" { ExternalVisible := 'False'} : Bool := FALSE;   // I806.0
      "I806.1" { ExternalVisible := 'False'} : Bool := FALSE;   // I806.1
      "I806.2" { ExternalVisible := 'False'} : Bool := FALSE;   // I806.2
      "I806.3" { ExternalVisible := 'False'} : Bool := FALSE;   // I806.3
      "I806.4" { ExternalVisible := 'False'} : Bool := FALSE;   // I806.4
      "I806.5" { ExternalVisible := 'False'} : Bool := FALSE;   // I806.5
      "I806.6" { ExternalVisible := 'False'} : Bool := FALSE;   // I806.6
      "I806.7" { ExternalVisible := 'False'} : Bool := FALSE;   // I806.7
      "I807.0" { ExternalVisible := 'False'} : Bool := FALSE;   // I807.0
      "I807.1" { ExternalVisible := 'False'} : Bool := FALSE;   // I807.1
      "I807.2" { ExternalVisible := 'False'} : Bool := FALSE;   // I807.2
      "I807.3" { ExternalVisible := 'False'} : Bool := FALSE;   // I807.3
      "I807.4" { ExternalVisible := 'False'} : Bool := FALSE;   // I807.4
      "I807.5" { ExternalVisible := 'False'} : Bool := FALSE;   // I807.5
      "I807.6" { ExternalVisible := 'False'} : Bool := FALSE;   // I807.6
      "I807.7" { ExternalVisible := 'False'} : Bool := FALSE;   // I807.7
      "I808.0" { ExternalVisible := 'False'} : Bool := FALSE;   // I808.0
      "I808.1" { ExternalVisible := 'False'} : Bool := FALSE;   // I808.1
      "I808.2" { ExternalVisible := 'False'} : Bool := FALSE;   // I808.2
      "I808.3" { ExternalVisible := 'False'} : Bool := FALSE;   // I808.3
      "I808.4" { ExternalVisible := 'False'} : Bool := FALSE;   // I808.4
      "I808.5" { ExternalVisible := 'False'} : Bool := FALSE;   // I808.5
      "I808.6" { ExternalVisible := 'False'} : Bool := FALSE;   // I808.6
      "I808.7" { ExternalVisible := 'False'} : Bool := FALSE;   // I808.7
      "I809.0" { ExternalVisible := 'False'} : Bool := FALSE;   // I809.0
      "I809.1" { ExternalVisible := 'False'} : Bool := FALSE;   // I809.1
      "I809.2" { ExternalVisible := 'False'} : Bool := FALSE;   // I809.2
      "I809.3" { ExternalVisible := 'False'} : Bool := FALSE;   // I809.3
      "I809.4" { ExternalVisible := 'False'} : Bool := FALSE;   // I809.4
      "I809.5" { ExternalVisible := 'False'} : Bool := FALSE;   // I809.5
      "I809.6" { ExternalVisible := 'False'} : Bool := FALSE;   // I809.6
      "I809.7" { ExternalVisible := 'False'} : Bool := FALSE;   // I809.7
      "I810.0" { ExternalVisible := 'False'} : Bool := FALSE;   // I810.0
      "I810.1" { ExternalVisible := 'False'} : Bool := FALSE;   // I810.1
      "I810.2" { ExternalVisible := 'False'} : Bool := FALSE;   // I810.2
      "I810.3" { ExternalVisible := 'False'} : Bool := FALSE;   // I810.3
      "I810.4" { ExternalVisible := 'False'} : Bool := FALSE;   // I810.4
      "I810.5" { ExternalVisible := 'False'} : Bool := FALSE;   // I810.5
      "I810.6" { ExternalVisible := 'False'} : Bool := FALSE;   // I810.6
      "I810.7" { ExternalVisible := 'False'} : Bool := FALSE;   // I810.7
      "I811.0" { ExternalVisible := 'False'} : Bool := FALSE;   // I811.0
      "I811.1" { ExternalVisible := 'False'} : Bool := FALSE;   // I811.1
      "I811.2" { ExternalVisible := 'False'} : Bool := FALSE;   // I811.2
      "I811.3" { ExternalVisible := 'False'} : Bool := FALSE;   // I811.3
      "I811.4" { ExternalVisible := 'False'} : Bool := FALSE;   // I811.4
      "I811.5" { ExternalVisible := 'False'} : Bool := FALSE;   // I811.5
      "I811.6" { ExternalVisible := 'False'} : Bool := FALSE;   // I811.6
      "I811.7" { ExternalVisible := 'False'} : Bool := FALSE;   // I811.7
      "I812.0" { ExternalVisible := 'False'} : Bool := FALSE;   // I812.0
      "I812.1" { ExternalVisible := 'False'} : Bool := FALSE;   // I812.1
      "I812.2" { ExternalVisible := 'False'} : Bool := FALSE;   // I812.2
      "I812.3" { ExternalVisible := 'False'} : Bool := FALSE;   // I812.3
      "I812.4" { ExternalVisible := 'False'} : Bool := FALSE;   // I812.4
      "I812.5" { ExternalVisible := 'False'} : Bool := FALSE;   // I812.5
      "I812.6" { ExternalVisible := 'False'} : Bool := FALSE;   // I812.6
      "I812.7" { ExternalVisible := 'False'} : Bool := FALSE;   // I812.7
      "I813.0" { ExternalVisible := 'False'} : Bool := FALSE;   // I813.0
      "I813.1" { ExternalVisible := 'False'} : Bool := FALSE;   // I813.1
      "I813.2" { ExternalVisible := 'False'} : Bool := FALSE;   // I813.2
      "I813.3" { ExternalVisible := 'False'} : Bool := FALSE;   // I813.3
      "I813.4" { ExternalVisible := 'False'} : Bool := FALSE;   // I813.4
      "I813.5" { ExternalVisible := 'False'} : Bool := FALSE;   // I813.5
      "I813.6" { ExternalVisible := 'False'} : Bool := FALSE;   // I813.6
      "I813.7" { ExternalVisible := 'False'} : Bool := FALSE;   // I813.7
      "I814.0" { ExternalVisible := 'False'} : Bool := FALSE;   // I814.0
      "I814.1" { ExternalVisible := 'False'} : Bool := FALSE;   // I814.1
      "I814.2" { ExternalVisible := 'False'} : Bool := FALSE;   // I814.2
      "I814.3" { ExternalVisible := 'False'} : Bool := FALSE;   // I814.3
      "I814.4" { ExternalVisible := 'False'} : Bool := FALSE;   // I814.4
      "I814.5" { ExternalVisible := 'False'} : Bool := FALSE;   // I814.5
      "I814.6" { ExternalVisible := 'False'} : Bool := FALSE;   // I814.6
      "I814.7" { ExternalVisible := 'False'} : Bool := FALSE;   // I814.7
      "I815.0" { ExternalVisible := 'False'} : Bool := FALSE;   // I815.0
      "I815.1" { ExternalVisible := 'False'} : Bool := FALSE;   // I815.1
      "I815.2" { ExternalVisible := 'False'} : Bool := FALSE;   // I815.2
      "I815.3" { ExternalVisible := 'False'} : Bool := FALSE;   // I815.3
      "I815.4" { ExternalVisible := 'False'} : Bool := FALSE;   // I815.4
      "I815.5" { ExternalVisible := 'False'} : Bool := FALSE;   // I815.5
      "I815.6" { ExternalVisible := 'False'} : Bool := FALSE;   // I815.6
      "I815.7" { ExternalVisible := 'False'} : Bool := FALSE;   // I815.7
      "I816.0" { ExternalVisible := 'False'} : Bool := FALSE;   // I816.0
      "I816.1" { ExternalVisible := 'False'} : Bool := FALSE;   // I816.1
      "I816.2" { ExternalVisible := 'False'} : Bool := FALSE;   // I816.2
      "I816.3" { ExternalVisible := 'False'} : Bool := FALSE;   // I816.3
      "I816.4" { ExternalVisible := 'False'} : Bool := FALSE;   // I816.4
      "I816.5" { ExternalVisible := 'False'} : Bool := FALSE;   // I816.5
      "I816.6" { ExternalVisible := 'False'} : Bool := FALSE;   // I816.6
      "I816.7" { ExternalVisible := 'False'} : Bool := FALSE;   // I816.7
      "I817.0" { ExternalVisible := 'False'} : Bool := FALSE;   // I817.0
      "I817.1" { ExternalVisible := 'False'} : Bool := FALSE;   // I817.1
      "I817.2" { ExternalVisible := 'False'} : Bool := FALSE;   // I817.2
      "I817.3" { ExternalVisible := 'False'} : Bool := FALSE;   // I817.3
      "I817.4" { ExternalVisible := 'False'} : Bool := FALSE;   // I817.4
      "I817.5" { ExternalVisible := 'False'} : Bool := FALSE;   // I817.5
      "I817.6" { ExternalVisible := 'False'} : Bool := FALSE;   // I817.6
      "I817.7" { ExternalVisible := 'False'} : Bool := FALSE;   // I817.7
      "I818.0" { ExternalVisible := 'False'} : Bool := FALSE;   // I818.0
      "I818.1" { ExternalVisible := 'False'} : Bool := FALSE;   // I818.1
      "I818.2" { ExternalVisible := 'False'} : Bool := FALSE;   // I818.2
      "I818.3" { ExternalVisible := 'False'} : Bool := FALSE;   // I818.3
      "I818.4" { ExternalVisible := 'False'} : Bool := FALSE;   // I818.4
      "I818.5" { ExternalVisible := 'False'} : Bool := FALSE;   // I818.5
      "I818.6" { ExternalVisible := 'False'} : Bool := FALSE;   // I818.6
      "I818.7" { ExternalVisible := 'False'} : Bool := FALSE;   // I818.7
      "I819.0" { ExternalVisible := 'False'} : Bool := FALSE;   // I819.0
      "I819.1" { ExternalVisible := 'False'} : Bool := FALSE;   // I819.1
      "I819.2" { ExternalVisible := 'False'} : Bool := FALSE;   // I819.2
      "I819.3" { ExternalVisible := 'False'} : Bool := FALSE;   // I819.3
      "I819.4" { ExternalVisible := 'False'} : Bool := FALSE;   // I819.4
      "I819.5" { ExternalVisible := 'False'} : Bool := FALSE;   // I819.5
      "I819.6" { ExternalVisible := 'False'} : Bool := FALSE;   // I819.6
      "I819.7" { ExternalVisible := 'False'} : Bool := FALSE;   // I819.7
      "I820.0" { ExternalVisible := 'False'} : Bool := FALSE;   // I820.0
      "I820.1" { ExternalVisible := 'False'} : Bool := FALSE;   // I820.1
      "I820.2" { ExternalVisible := 'False'} : Bool := FALSE;   // I820.2
      "I820.3" { ExternalVisible := 'False'} : Bool := FALSE;   // I820.3
      "I820.4" { ExternalVisible := 'False'} : Bool := FALSE;   // I820.4
      "I820.5" { ExternalVisible := 'False'} : Bool := FALSE;   // I820.5
      "I820.6" { ExternalVisible := 'False'} : Bool := FALSE;   // I820.6
      "I820.7" { ExternalVisible := 'False'} : Bool := FALSE;   // I820.7
      "I821.0" { ExternalVisible := 'False'} : Bool := FALSE;   // I821.0
      "I821.1" { ExternalVisible := 'False'} : Bool := FALSE;   // I821.1
      "I821.2" { ExternalVisible := 'False'} : Bool := FALSE;   // I821.2
      "I821.3" { ExternalVisible := 'False'} : Bool := FALSE;   // I821.3
      "I821.4" { ExternalVisible := 'False'} : Bool := FALSE;   // I821.4
      "I821.5" { ExternalVisible := 'False'} : Bool := FALSE;   // I821.5
      "I821.6" { ExternalVisible := 'False'} : Bool := FALSE;   // I821.6
      "I821.7" { ExternalVisible := 'False'} : Bool := FALSE;   // I821.7
      "I822.0" { ExternalVisible := 'False'} : Bool := FALSE;   // I822.0
      "I822.1" { ExternalVisible := 'False'} : Bool := FALSE;   // I822.1
      "I822.2" { ExternalVisible := 'False'} : Bool := FALSE;   // I822.2
      "I822.3" { ExternalVisible := 'False'} : Bool := FALSE;   // I822.3
      "I822.4" { ExternalVisible := 'False'} : Bool := FALSE;   // I822.4
      "I822.5" { ExternalVisible := 'False'} : Bool := FALSE;   // I822.5
      "I822.6" { ExternalVisible := 'False'} : Bool := FALSE;   // I822.6
      "I822.7" { ExternalVisible := 'False'} : Bool := FALSE;   // I822.7
      "I823.0" { ExternalVisible := 'False'} : Bool := FALSE;   // I823.0
      "I823.1" { ExternalVisible := 'False'} : Bool := FALSE;   // I823.1
      "I823.2" { ExternalVisible := 'False'} : Bool := FALSE;   // I823.2
      "I823.3" { ExternalVisible := 'False'} : Bool := FALSE;   // I823.3
      "I823.4" { ExternalVisible := 'False'} : Bool := FALSE;   // I823.4
      "I823.5" { ExternalVisible := 'False'} : Bool := FALSE;   // I823.5
      "I823.6" { ExternalVisible := 'False'} : Bool := FALSE;   // I823.6
      "I823.7" { ExternalVisible := 'False'} : Bool := FALSE;   // I823.7
      "I824.0" { ExternalVisible := 'False'} : Bool := FALSE;   // I824.0
      "I824.1" { ExternalVisible := 'False'} : Bool := FALSE;   // I824.1
      "I824.2" { ExternalVisible := 'False'} : Bool := FALSE;   // I824.2
      "I824.3" { ExternalVisible := 'False'} : Bool := FALSE;   // I824.3
      "I824.4" { ExternalVisible := 'False'} : Bool := FALSE;   // I824.4
      "I824.5" { ExternalVisible := 'False'} : Bool := FALSE;   // I824.5
      "I824.6" { ExternalVisible := 'False'} : Bool := FALSE;   // I824.6
      "I824.7" { ExternalVisible := 'False'} : Bool := FALSE;   // I824.7
      "I825.0" { ExternalVisible := 'False'} : Bool := FALSE;   // I825.0
      "I825.1" { ExternalVisible := 'False'} : Bool := FALSE;   // I825.1
      "I825.2" { ExternalVisible := 'False'} : Bool := FALSE;   // I825.2
      "I825.3" { ExternalVisible := 'False'} : Bool := FALSE;   // I825.3
      "I825.4" { ExternalVisible := 'False'} : Bool := FALSE;   // I825.4
      "I825.5" { ExternalVisible := 'False'} : Bool := FALSE;   // I825.5
      "I825.6" { ExternalVisible := 'False'} : Bool := FALSE;   // I825.6
      "I825.7" { ExternalVisible := 'False'} : Bool := FALSE;   // I825.7
      "I826.0" { ExternalVisible := 'False'} : Bool := FALSE;   // I826.0
      "I826.1" { ExternalVisible := 'False'} : Bool := FALSE;   // I826.1
      "I826.2" { ExternalVisible := 'False'} : Bool := FALSE;   // I826.2
      "I826.3" { ExternalVisible := 'False'} : Bool := FALSE;   // I826.3
      "I826.4" { ExternalVisible := 'False'} : Bool := FALSE;   // I826.4
      "I826.5" { ExternalVisible := 'False'} : Bool := FALSE;   // I826.5
      "I826.6" { ExternalVisible := 'False'} : Bool := FALSE;   // I826.6
      "I826.7" { ExternalVisible := 'False'} : Bool := FALSE;   // I826.7
      "I827.0" { ExternalVisible := 'False'} : Bool := FALSE;   // I827.0
      "I827.1" { ExternalVisible := 'False'} : Bool := FALSE;   // I827.1
      "I827.2" { ExternalVisible := 'False'} : Bool := FALSE;   // I827.2
      "I827.3" { ExternalVisible := 'False'} : Bool := FALSE;   // I827.3
      "I827.4" { ExternalVisible := 'False'} : Bool := FALSE;   // I827.4
      "I827.5" { ExternalVisible := 'False'} : Bool := FALSE;   // I827.5
      "I827.6" { ExternalVisible := 'False'} : Bool := FALSE;   // I827.6
      "I827.7" { ExternalVisible := 'False'} : Bool := FALSE;   // I827.7
      "I828.0" { ExternalVisible := 'False'} : Bool := FALSE;   // I828.0
      "I828.1" { ExternalVisible := 'False'} : Bool := FALSE;   // I828.1
      "I828.2" { ExternalVisible := 'False'} : Bool := FALSE;   // I828.2
      "I828.3" { ExternalVisible := 'False'} : Bool := FALSE;   // I828.3
      "I828.4" { ExternalVisible := 'False'} : Bool := FALSE;   // I828.4
      "I828.5" { ExternalVisible := 'False'} : Bool := FALSE;   // I828.5
      "I828.6" { ExternalVisible := 'False'} : Bool := FALSE;   // I828.6
      "I828.7" { ExternalVisible := 'False'} : Bool := FALSE;   // I828.7
      "I829.0" { ExternalVisible := 'False'} : Bool := FALSE;   // I829.0
      "I829.1" { ExternalVisible := 'False'} : Bool := FALSE;   // I829.1
      "I829.2" { ExternalVisible := 'False'} : Bool := FALSE;   // I829.2
      "I829.3" { ExternalVisible := 'False'} : Bool := FALSE;   // I829.3
      "I829.4" { ExternalVisible := 'False'} : Bool := FALSE;   // I829.4
      "I829.5" { ExternalVisible := 'False'} : Bool := FALSE;   // I829.5
      "I829.6" { ExternalVisible := 'False'} : Bool := FALSE;   // I829.6
      "I829.7" { ExternalVisible := 'False'} : Bool := FALSE;   // I829.7
      "I830.0" { ExternalVisible := 'False'} : Bool := FALSE;   // I830.0
      "I830.1" { ExternalVisible := 'False'} : Bool := FALSE;   // I830.1
      "I830.2" { ExternalVisible := 'False'} : Bool := FALSE;   // I830.2
      "I830.3" { ExternalVisible := 'False'} : Bool := FALSE;   // I830.3
      "I830.4" { ExternalVisible := 'False'} : Bool := FALSE;   // I830.4
